LIN {X 0,Y 525.761,Z 1147.71,A -85,B 0,C 180,E1 17885.507,E2 17885.507} C_VEL
LIN {X 0,Y 527.869,Z 1135.72,A -85,B 0,C 180,E1 17883.205,E2 17883.205} C_VEL
LIN {X 0,Y 530.322,Z 1123.021,A -85,B 0,C 180,E1 17881.027,E2 17881.027} C_VEL
LIN {X 0,Y 533.766,Z 1106.397,A -85,B 0,C 180,E1 17878.491,E2 17878.491} C_VEL
LIN {X 0,Y 537.469,Z 1088.541,A -85,B 0,C 180,E1 17876.14,E2 17876.14} C_VEL
LIN {X 0,Y 540.914,Z 1072.555,A -85,B 0,C 180,E1 17874.259,E2 17874.259} C_VEL
LIN {X 0,Y 544.546,Z 1055.798,A -85,B 0,C 180,E1 17872.489,E2 17872.489} C_VEL
LIN {X 0,Y 549.152,Z 1034.672,A -85,B 0,C 180,E1 17870.505,E2 17870.505} C_VEL
LIN {X 0,Y 553.58,Z 1013.13,A -85,B 0,C 180,E1 17868.757,E2 17868.757} C_VEL
LIN {X 0,Y 557.256,Z 994.74,A -85,B 0,C 180,E1 17867.434,E2 17867.434} C_VEL
LIN {X 0,Y 560.832,Z 975.985,A -85,B 0,C 180,E1 17866.232,E2 17866.232} C_VEL
LIN {X 0,Y 564.294,Z 956.689,A -85,B 0,C 180,E1 17865.135,E2 17865.135} C_VEL
LIN {X 0,Y 568.047,Z 934.279,A -85,B 0,C 180,E1 17864.025,E2 17864.025} C_VEL
LIN {X 0,Y 572.034,Z 907.383,A -85,B 0,C 180,E1 17862.914,E2 17862.914} C_VEL
LIN {X 0,Y 574.908,Z 884.853,A -85,B 0,C 180,E1 17862.151,E2 17862.151} C_VEL
LIN {X 0,Y 577.234,Z 863.544,A -85,B 0,C 180,E1 17861.557,E2 17861.557} C_VEL
LIN {X 0,Y 579.186,Z 841.987,A -85,B 0,C 180,E1 17861.078,E2 17861.078} C_VEL
LIN {X 0,Y 580.867,Z 815.756,A -85,B 0,C 180,E1 17860.629,E2 17860.629} C_VEL
LIN {X 0,Y 589.677,Z 592.24,A -85,B 0,C 180,E1 17857.327,E2 17857.327} C_VEL
LIN {X 0,Y 595.841,Z 445.382,A -85,B 0,C 180,E1 17855.112,E2 17855.112} C_VEL
LIN {X 0,Y 585.604,Z 429.266,A -85,B 0,C 180,E1 17853.178,E2 17853.178} C_VEL
LIN {X 0,Y 575.982,Z 415.554,A -85,B 0,C 180,E1 17851.211,E2 17851.211} C_VEL
LIN {X 0,Y 566.461,Z 402.539,A -85,B 0,C 180,E1 17849.069,E2 17849.069} C_VEL
LIN {X 0,Y 561.316,Z 396.051,A -85,B 0,C 180,E1 17847.821,E2 17847.821} C_VEL
LIN {X 0,Y 556.973,Z 390.44,A -85,B 0,C 180,E1 17846.696,E2 17846.696} C_VEL
LIN {X 0,Y 552.471,Z 384.765,A -85,B 0,C 180,E1 17845.458,E2 17845.458} C_VEL
LIN {X 0,Y 548.916,Z 380.538,A -85,B 0,C 180,E1 17844.425,E2 17844.425} C_VEL
LIN {X 0,Y 544.6,Z 375.283,A -85,B 0,C 180,E1 17843.078,E2 17843.078} C_VEL
LIN {X 0,Y 541.358,Z 372.099,A -85,B 0,C 180,E1 17842.021,E2 17842.021} C_VEL
LIN {X 0,Y 539.707,Z 369.279,A -85,B 0,C 180,E1 17841.406,E2 17841.406} C_VEL
LIN {X 0,Y 536.376,Z 366.847,A -85,B 0,C 180,E1 17840.231,E2 17840.231} C_VEL
LIN {X 0,Y 534.263,Z 363.307,A -85,B 0,C 180,E1 17839.345,E2 17839.345} C_VEL
LIN {X 0,Y 533.757,Z 362.736,A -85,B 0,C 180,E1 17839.137,E2 17839.137} C_VEL
LIN {X 0,Y 530.459,Z 360.54,A -85,B 0,C 180,E1 17837.78,E2 17837.78} C_VEL
LIN {X 0,Y 528.468,Z 357.561,A -85,B 0,C 180,E1 17836.802,E2 17836.802} C_VEL
LIN {X 0,Y 527.857,Z 356.011,A -85,B 0,C 180,E1 17836.451,E2 17836.451} C_VEL
LIN {X 0,Y 524.184,Z 354.141,A -85,B 0,C 180,E1 17834.584,E2 17834.584} C_VEL
LIN {X 0,Y 522.044,Z 350.897,A -85,B 0,C 180,E1 17833.175,E2 17833.175} C_VEL
LIN {X 0,Y 521.643,Z 349.211,A -85,B 0,C 180,E1 17832.735,E2 17832.735} C_VEL
LIN {X 0,Y 521.673,Z 349.223,A -85,B 0,C 180,E1 17829.376,E2 17829.376} C_VEL
LIN {X 0,Y 521.662,Z 349.19,A -85,B 0,C 180,E1 17826.272,E2 17826.272} C_VEL
LIN {X 0,Y 521.662,Z 349.252,A -85,B 0,C 180,E1 17822.857,E2 17822.857} C_VEL
LIN {X 0,Y 521.731,Z 349.183,A -85,B 0,C 180,E1 17819.561,E2 17819.561} C_VEL
LIN {X 0,Y 521.66,Z 349.21,A -85,B 0,C 180,E1 17816.263,E2 17816.263} C_VEL
LIN {X 0,Y 521.695,Z 349.269,A -85,B 0,C 180,E1 17812.954,E2 17812.954} C_VEL
LIN {X 0,Y 522.394,Z 351.72,A -85,B 0,C 180,E1 17812.355,E2 17812.355} C_VEL
LIN {X 0,Y 524.741,Z 354.555,A -85,B 0,C 180,E1 17810.9,E2 17810.9} C_VEL
LIN {X 0,Y 528.048,Z 356.193,A -85,B 0,C 180,E1 17809.25,E2 17809.25} C_VEL
LIN {X 0,Y 529.406,Z 359.289,A -85,B 0,C 180,E1 17808.506,E2 17808.506} C_VEL
LIN {X 0,Y 532.127,Z 361.898,A -85,B 0,C 180,E1 17807.3,E2 17807.3} C_VEL
LIN {X 0,Y 534.16,Z 363.105,A -85,B 0,C 180,E1 17806.496,E2 17806.496} C_VEL
LIN {X 0,Y 536.193,Z 366.523,A -85,B 0,C 180,E1 17805.64,E2 17805.64} C_VEL
LIN {X 0,Y 539.324,Z 369.091,A -85,B 0,C 180,E1 17804.516,E2 17804.516} C_VEL
LIN {X 0,Y 540.125,Z 369.854,A -85,B 0,C 180,E1 17804.236,E2 17804.236} C_VEL
LIN {X 0,Y 542.762,Z 373.729,A -85,B 0,C 180,E1 17803.298,E2 17803.298} C_VEL
LIN {X 0,Y 545.709,Z 376.231,A -85,B 0,C 180,E1 17802.375,E2 17802.375} C_VEL
LIN {X 0,Y 548.797,Z 380.377,A -85,B 0,C 180,E1 17801.407,E2 17801.407} C_VEL
LIN {X 0,Y 551.115,Z 382.496,A -85,B 0,C 180,E1 17800.746,E2 17800.746} C_VEL
LIN {X 0,Y 554.639,Z 386.927,A -85,B 0,C 180,E1 17799.749,E2 17799.749} C_VEL
LIN {X 0,Y 556.439,Z 388.927,A -85,B 0,C 180,E1 17799.268,E2 17799.268} C_VEL
LIN {X 0,Y 560.51,Z 393.596,A -85,B 0,C 180,E1 17798.219,E2 17798.219} C_VEL
LIN {X 0,Y 564.909,Z 399.046,A -85,B 0,C 180,E1 17797.138,E2 17797.138} C_VEL
LIN {X 0,Y 574.234,Z 410.747,A -85,B 0,C 180,E1 17795.023,E2 17795.023} C_VEL
LIN {X 0,Y 581.384,Z 420.611,A -85,B 0,C 180,E1 17793.521,E2 17793.521} C_VEL
LIN {X 0,Y 590.334,Z 433.608,A -85,B 0,C 180,E1 17791.772,E2 17791.772} C_VEL
LIN {X 0,Y 595.87,Z 442.641,A -85,B 0,C 180,E1 17790.739,E2 17790.739} C_VEL
LIN {X 0,Y 586.827,Z 657.464,A -85,B 0,C 180,E1 17787.527,E2 17787.527} C_VEL
LIN {X 0,Y 580.388,Z 818.126,A -85,B 0,C 180,E1 17785.144,E2 17785.144} C_VEL
LIN {X 0,Y 578.549,Z 843.265,A -85,B 0,C 180,E1 17784.67,E2 17784.67} C_VEL
LIN {X 0,Y 575.726,Z 870.858,A -85,B 0,C 180,E1 17783.958,E2 17783.958} C_VEL
LIN {X 0,Y 573.031,Z 892.591,A -85,B 0,C 180,E1 17783.253,E2 17783.253} C_VEL
LIN {X 0,Y 570.192,Z 912.82,A -85,B 0,C 180,E1 17782.471,E2 17782.471} C_VEL
LIN {X 0,Y 566.949,Z 933.521,A -85,B 0,C 180,E1 17781.539,E2 17781.539} C_VEL
LIN {X 0,Y 563.55,Z 953.219,A -85,B 0,C 180,E1 17780.521,E2 17780.521} C_VEL
LIN {X 0,Y 561.609,Z 960.127,A -85,B 0,C 180,E1 17780.208,E2 17780.208} C_VEL
LIN {X 0,Y 553.835,Z 977.712,A -85,B 0,C 180,E1 17779.574,E2 17779.574} C_VEL
LIN {X 0,Y 551.762,Z 984.148,A -85,B 0,C 180,E1 17779.207,E2 17779.207} C_VEL
LIN {X 0,Y 547.898,Z 1002.415,A -85,B 0,C 180,E1 17777.887,E2 17777.887} C_VEL
LIN {X 0,Y 543.458,Z 1022.804,A -85,B 0,C 180,E1 17776.228,E2 17776.228} C_VEL
LIN {X 0,Y 538.244,Z 1045.707,A -85,B 0,C 180,E1 17774.074,E2 17774.074} C_VEL
LIN {X 0,Y 534.354,Z 1062.517,A -85,B 0,C 180,E1 17772.274,E2 17772.274} C_VEL
LIN {X 0,Y 530.736,Z 1078.224,A -85,B 0,C 180,E1 17770.396,E2 17770.396} C_VEL
LIN {X 0,Y 526.924,Z 1095.053,A -85,B 0,C 180,E1 17768.145,E2 17768.145} C_VEL
LIN {X 0,Y 523.166,Z 1112.322,A -85,B 0,C 180,E1 17765.493,E2 17765.493} C_VEL
LIN {X 0,Y 520.447,Z 1125.546,A -85,B 0,C 180,E1 17763.198,E2 17763.198} C_VEL
LIN {X 0,Y 518.304,Z 1136.869,A -85,B 0,C 180,E1 17761.002,E2 17761.002} C_VEL
LIN {X 0,Y 516.4,Z 1148.029,A -85,B 0,C 180,E1 17758.571,E2 17758.571} C_VEL
LIN {X 0,Y 514.548,Z 1160.441,A -85,B 0,C 180,E1 17755.432,E2 17755.432} C_VEL
LIN {X 0,Y 513.475,Z 1169.219,A -85,B 0,C 180,E1 17752.799,E2 17752.799} C_VEL
LIN {X 0,Y 512.794,Z 1176.005,A -85,B 0,C 180,E1 17750.427,E2 17750.427} C_VEL
LIN {X 0,Y 512.354,Z 1181.938,A -85,B 0,C 180,E1 17747.959,E2 17747.959} C_VEL
LIN {X 0,Y 512.062,Z 1187.545,A -85,B 0,C 180,E1 17745.052,E2 17745.052} C_VEL
LIN {X 0,Y 511.941,Z 1191.578,A -85,B 0,C 180,E1 17742.062,E2 17742.062} C_VEL
LIN {X 0,Y 511.916,Z 1193.749,A -85,B 0,C 180,E1 17739.556,E2 17739.556} C_VEL
LIN {X 0,Y 511.911,Z 1194.759,A -85,B 0,C 180,E1 17737.181,E2 17737.181} C_VEL
LIN {X 0,Y 511.902,Z 1194.8,A -85,B 0,C 180,E1 17734.93,E2 17734.93} C_VEL
LIN {X 0,Y 511.914,Z 1193.884,A -85,B 0,C 180,E1 17732.574,E2 17732.574} C_VEL
LIN {X 0,Y 511.948,Z 1191.845,A -85,B 0,C 180,E1 17730.111,E2 17730.111} C_VEL
LIN {X 0,Y 512.038,Z 1188.251,A -85,B 0,C 180,E1 17727.313,E2 17727.313} C_VEL
LIN {X 0,Y 512.321,Z 1182.436,A -85,B 0,C 180,E1 17724.175,E2 17724.175} C_VEL
LIN {X 0,Y 512.76,Z 1176.29,A -85,B 0,C 180,E1 17721.59,E2 17721.59} C_VEL
LIN {X 0,Y 513.474,Z 1169.223,A -85,B 0,C 180,E1 17719.112,E2 17719.112} C_VEL
LIN {X 0,Y 514.472,Z 1160.962,A -85,B 0,C 180,E1 17716.627,E2 17716.627} C_VEL
LIN {X 0,Y 516.231,Z 1149.055,A -85,B 0,C 180,E1 17713.573,E2 17713.573} C_VEL
LIN {X 0,Y 518.247,Z 1137.167,A -85,B 0,C 180,E1 17710.97,E2 17710.97} C_VEL
LIN {X 0,Y 520.43,Z 1125.525,A -85,B 0,C 180,E1 17708.708,E2 17708.708} C_VEL
LIN {X 0,Y 523.27,Z 1111.869,A -85,B 0,C 180,E1 17706.342,E2 17706.342} C_VEL
LIN {X 0,Y 527.274,Z 1093.391,A -85,B 0,C 180,E1 17703.536,E2 17703.536} C_VEL
LIN {X 0,Y 530.909,Z 1077.464,A -85,B 0,C 180,E1 17701.421,E2 17701.421} C_VEL
LIN {X 0,Y 534.559,Z 1061.663,A -85,B 0,C 180,E1 17699.542,E2 17699.542} C_VEL
LIN {X 0,Y 539.256,Z 1041.498,A -85,B 0,C 180,E1 17697.409,E2 17697.409} C_VEL
LIN {X 0,Y 544.119,Z 1019.613,A -85,B 0,C 180,E1 17695.413,E2 17695.413} C_VEL
LIN {X 0,Y 548.064,Z 1001.544,A -85,B 0,C 180,E1 17693.959,E2 17693.959} C_VEL
LIN {X 0,Y 551.937,Z 983.052,A -85,B 0,C 180,E1 17692.635,E2 17692.635} C_VEL
LIN {X 0,Y 555.697,Z 964.008,A -85,B 0,C 180,E1 17691.43,E2 17691.43} C_VEL
LIN {X 0,Y 560.006,Z 940.548,A -85,B 0,C 180,E1 17690.134,E2 17690.134} C_VEL
LIN {X 0,Y 563.885,Z 915.971,A -85,B 0,C 180,E1 17688.998,E2 17688.998} C_VEL
LIN {X 0,Y 566.87,Z 895.119,A -85,B 0,C 180,E1 17688.184,E2 17688.184} C_VEL
LIN {X 0,Y 569.491,Z 874.162,A -85,B 0,C 180,E1 17687.494,E2 17687.494} C_VEL
LIN {X 0,Y 571.773,Z 852.476,A -85,B 0,C 180,E1 17686.905,E2 17686.905} C_VEL
LIN {X 0,Y 574.089,Z 825.329,A -85,B 0,C 180,E1 17686.335,E2 17686.335} C_VEL
LIN {X 0,Y 576.018,Z 780.91,A -85,B 0,C 180,E1 17685.663,E2 17685.663} C_VEL
LIN {X 0,Y 584.231,Z 560.655,A -85,B 0,C 180,E1 17682.446,E2 17682.446} C_VEL
LIN {X 0,Y 588.645,Z 446.135,A -85,B 0,C 180,E1 17680.742,E2 17680.742} C_VEL
LIN {X 0,Y 571.02,Z 420.614,A -85,B 0,C 180,E1 17677.734,E2 17677.734} C_VEL
LIN {X 0,Y 561.488,Z 408.03,A -85,B 0,C 180,E1 17675.96,E2 17675.96} C_VEL
LIN {X 0,Y 552.936,Z 397.243,A -85,B 0,C 180,E1 17674.253,E2 17674.253} C_VEL
LIN {X 0,Y 548.26,Z 391.475,A -85,B 0,C 180,E1 17673.264,E2 17673.264} C_VEL
LIN {X 0,Y 544.255,Z 386.546,A -85,B 0,C 180,E1 17672.381,E2 17672.381} C_VEL
LIN {X 0,Y 539.839,Z 381.182,A -85,B 0,C 180,E1 17671.364,E2 17671.364} C_VEL
LIN {X 0,Y 536.158,Z 376.858,A -85,B 0,C 180,E1 17670.482,E2 17670.482} C_VEL
LIN {X 0,Y 534.966,Z 375.343,A -85,B 0,C 180,E1 17670.184,E2 17670.184} C_VEL
LIN {X 0,Y 531.495,Z 371.631,A -85,B 0,C 180,E1 17669.315,E2 17669.315} C_VEL
LIN {X 0,Y 529.9,Z 369.383,A -85,B 0,C 180,E1 17668.885,E2 17668.885} C_VEL
LIN {X 0,Y 526.557,Z 366.145,A -85,B 0,C 180,E1 17668.003,E2 17668.003} C_VEL
LIN {X 0,Y 524.719,Z 363.213,A -85,B 0,C 180,E1 17667.461,E2 17667.461} C_VEL
LIN {X 0,Y 521.414,Z 360.538,A -85,B 0,C 180,E1 17666.54,E2 17666.54} C_VEL
LIN {X 0,Y 519.476,Z 357.042,A -85,B 0,C 180,E1 17665.908,E2 17665.908} C_VEL
LIN {X 0,Y 515.824,Z 354.574,A -85,B 0,C 180,E1 17664.814,E2 17664.814} C_VEL
LIN {X 0,Y 514.112,Z 351.727,A -85,B 0,C 180,E1 17664.212,E2 17664.212} C_VEL
LIN {X 0,Y 513.765,Z 350.215,A -85,B 0,C 180,E1 17664.017,E2 17664.017} C_VEL
LIN {X 0,Y 513.798,Z 350.151,A -85,B 0,C 180,E1 17660.625,E2 17660.625} C_VEL
LIN {X 0,Y 513.787,Z 350.233,A -85,B 0,C 180,E1 17657.15,E2 17657.15} C_VEL
LIN {X 0,Y 513.745,Z 350.152,A -85,B 0,C 180,E1 17653.736,E2 17653.736} C_VEL
LIN {X 0,Y 513.79,Z 350.234,A -85,B 0,C 180,E1 17650.314,E2 17650.314} C_VEL
LIN {X 0,Y 513.767,Z 350.234,A -85,B 0,C 180,E1 17646.999,E2 17646.999} C_VEL
LIN {X 0,Y 513.743,Z 350.238,A -85,B 0,C 180,E1 17643.571,E2 17643.571} C_VEL
LIN {X 0,Y 513.796,Z 350.226,A -85,B 0,C 180,E1 17640.223,E2 17640.223} C_VEL
LIN {X 0,Y 513.747,Z 350.231,A -85,B 0,C 180,E1 17636.876,E2 17636.876} C_VEL
LIN {X 0,Y 513.731,Z 350.234,A -85,B 0,C 180,E1 17633.406,E2 17633.406} C_VEL
LIN {X 0,Y 513.788,Z 350.224,A -85,B 0,C 180,E1 17630.139,E2 17630.139} C_VEL
LIN {X 0,Y 513.716,Z 350.164,A -85,B 0,C 180,E1 17626.837,E2 17626.837} C_VEL
LIN {X 0,Y 513.721,Z 350.242,A -85,B 0,C 180,E1 17623.256,E2 17623.256} C_VEL
LIN {X 0,Y 513.803,Z 350.41,A -85,B 0,C 180,E1 17622.034,E2 17622.034} C_VEL
LIN {X 0,Y 514.804,Z 353.275,A -85,B 0,C 180,E1 17621.631,E2 17621.631} C_VEL
LIN {X 0,Y 517.159,Z 355.808,A -85,B 0,C 180,E1 17620.87,E2 17620.87} C_VEL
LIN {X 0,Y 519.5,Z 357.171,A -85,B 0,C 180,E1 17620.185,E2 17620.185} C_VEL
LIN {X 0,Y 521.376,Z 360.616,A -85,B 0,C 180,E1 17619.571,E2 17619.571} C_VEL
LIN {X 0,Y 524.285,Z 363.051,A -85,B 0,C 180,E1 17618.755,E2 17618.755} C_VEL
LIN {X 0,Y 525.119,Z 363.758,A -85,B 0,C 180,E1 17618.527,E2 17618.527} C_VEL
LIN {X 0,Y 527.678,Z 367.626,A -85,B 0,C 180,E1 17617.788,E2 17617.788} C_VEL
LIN {X 0,Y 530.678,Z 370.269,A -85,B 0,C 180,E1 17617.015,E2 17617.015} C_VEL
LIN {X 0,Y 533.824,Z 374.393,A -85,B 0,C 180,E1 17616.194,E2 17616.194} C_VEL
LIN {X 0,Y 535.842,Z 376.372,A -85,B 0,C 180,E1 17615.703,E2 17615.703} C_VEL
LIN {X 0,Y 539.468,Z 380.812,A -85,B 0,C 180,E1 17614.826,E2 17614.826} C_VEL
LIN {X 0,Y 548.179,Z 392.031,A -85,B 0,C 180,E1 17612.841,E2 17612.841} C_VEL
LIN {X 0,Y 557.613,Z 404.61,A -85,B 0,C 180,E1 17610.867,E2 17610.867} C_VEL
LIN {X 0,Y 568.004,Z 419.104,A -85,B 0,C 180,E1 17608.862,E2 17608.862} C_VEL
LIN {X 0,Y 578.642,Z 434.507,A -85,B 0,C 180,E1 17606.963,E2 17606.963} C_VEL
LIN {X 0,Y 588.727,Z 449.63,A -85,B 0,C 180,E1 17605.282,E2 17605.282} C_VEL
LIN {X 0,Y 580.428,Z 665.627,A -85,B 0,C 180,E1 17602.1,E2 17602.1} C_VEL
LIN {X 0,Y 574.396,Z 825.945,A -85,B 0,C 180,E1 17599.753,E2 17599.753} C_VEL
LIN {X 0,Y 572.587,Z 850.931,A -85,B 0,C 180,E1 17599.291,E2 17599.291} C_VEL
LIN {X 0,Y 569.74,Z 879.117,A -85,B 0,C 180,E1 17598.579,E2 17598.579} C_VEL
LIN {X 0,Y 567.081,Z 900.684,A -85,B 0,C 180,E1 17597.891,E2 17597.891} C_VEL
LIN {X 0,Y 564.224,Z 921.047,A -85,B 0,C 180,E1 17597.117,E2 17597.117} C_VEL
LIN {X 0,Y 560.996,Z 941.562,A -85,B 0,C 180,E1 17596.207,E2 17596.207} C_VEL
LIN {X 0,Y 556.997,Z 964.706,A -85,B 0,C 180,E1 17595.014,E2 17595.014} C_VEL
LIN {X 0,Y 552.173,Z 989.793,A -85,B 0,C 180,E1 17593.481,E2 17593.481} C_VEL
LIN {X 0,Y 548.272,Z 1008.652,A -85,B 0,C 180,E1 17592.154,E2 17592.154} C_VEL
LIN {X 0,Y 544.322,Z 1026.988,A -85,B 0,C 180,E1 17590.701,E2 17590.701} C_VEL
LIN {X 0,Y 540.247,Z 1045.394,A -85,B 0,C 180,E1 17589.064,E2 17589.064} C_VEL
LIN {X 0,Y 535.329,Z 1067.372,A -85,B 0,C 180,E1 17586.839,E2 17586.839} C_VEL
LIN {X 0,Y 531.263,Z 1085.188,A -85,B 0,C 180,E1 17584.769,E2 17584.769} C_VEL
LIN {X 0,Y 528.055,Z 1099.499,A -85,B 0,C 180,E1 17582.918,E2 17582.918} C_VEL
LIN {X 0,Y 525.032,Z 1113.285,A -85,B 0,C 180,E1 17580.944,E2 17580.944} C_VEL
LIN {X 0,Y 522.122,Z 1127.161,A -85,B 0,C 180,E1 17578.73,E2 17578.73} C_VEL
LIN {X 0,Y 519.004,Z 1143.111,A -85,B 0,C 180,E1 17575.811,E2 17575.811} C_VEL
LIN {X 0,Y 516.93,Z 1154.734,A -85,B 0,C 180,E1 17573.361,E2 17573.361} C_VEL
LIN {X 0,Y 515.375,Z 1164.513,A -85,B 0,C 180,E1 17571.034,E2 17571.034} C_VEL
LIN {X 0,Y 514.148,Z 1173.506,A -85,B 0,C 180,E1 17568.599,E2 17568.599} C_VEL
LIN {X 0,Y 513.09,Z 1183.01,A -85,B 0,C 180,E1 17565.601,E2 17565.601} C_VEL
LIN {X 0,Y 512.439,Z 1190.44,A -85,B 0,C 180,E1 17562.676,E2 17562.676} C_VEL
LIN {X 0,Y 512.138,Z 1195.692,A -85,B 0,C 180,E1 17560.121,E2 17560.121} C_VEL
LIN {X 0,Y 511.987,Z 1199.677,A -85,B 0,C 180,E1 17557.632,E2 17557.632} C_VEL
LIN {X 0,Y 511.926,Z 1202.768,A -85,B 0,C 180,E1 17554.93,E2 17554.93} C_VEL
LIN {X 0,Y 511.91,Z 1204.622,A -85,B 0,C 180,E1 17551.903,E2 17551.903} C_VEL
LIN {X 0,Y 511.897,Z 1204.871,A -85,B 0,C 180,E1 17549.329,E2 17549.329} C_VEL
LIN {X 0,Y 511.916,Z 1204.032,A -85,B 0,C 180,E1 17546.865,E2 17546.865} C_VEL
LIN {X 0,Y 511.936,Z 1202.085,A -85,B 0,C 180,E1 17544.396,E2 17544.396} C_VEL
LIN {X 0,Y 512.01,Z 1199.038,A -85,B 0,C 180,E1 17541.918,E2 17541.918} C_VEL
LIN {X 0,Y 512.197,Z 1194.454,A -85,B 0,C 180,E1 17539.199,E2 17539.199} C_VEL
LIN {X 0,Y 512.7,Z 1187.27,A -85,B 0,C 180,E1 17536.006,E2 17536.006} C_VEL
LIN {X 0,Y 513.354,Z 1180.209,A -85,B 0,C 180,E1 17533.479,E2 17533.479} C_VEL
LIN {X 0,Y 514.301,Z 1172.293,A -85,B 0,C 180,E1 17531.055,E2 17531.055} C_VEL
LIN {X 0,Y 515.578,Z 1163.145,A -85,B 0,C 180,E1 17528.618,E2 17528.618} C_VEL
LIN {X 0,Y 517.641,Z 1150.764,A -85,B 0,C 180,E1 17525.746,E2 17525.746} C_VEL
LIN {X 0,Y 520.149,Z 1136.988,A -85,B 0,C 180,E1 17523.022,E2 17523.022} C_VEL
LIN {X 0,Y 522.702,Z 1124.358,A -85,B 0,C 180,E1 17520.805,E2 17520.805} C_VEL
LIN {X 0,Y 525.619,Z 1110.662,A -85,B 0,C 180,E1 17518.665,E2 17518.665} C_VEL
LIN {X 0,Y 529.598,Z 1092.624,A -85,B 0,C 180,E1 17516.155,E2 17516.155} C_VEL
LIN {X 0,Y 533.769,Z 1073.974,A -85,B 0,C 180,E1 17513.905,E2 17513.905} C_VEL
LIN {X 0,Y 537.501,Z 1057.5,A -85,B 0,C 180,E1 17512.13,E2 17512.13} C_VEL
LIN {X 0,Y 541.483,Z 1039.846,A -85,B 0,C 180,E1 17510.428,E2 17510.428} C_VEL
LIN {X 0,Y 546.452,Z 1017.438,A -85,B 0,C 180,E1 17508.52,E2 17508.52} C_VEL
LIN {X 0,Y 551.03,Z 995.494,A -85,B 0,C 180,E1 17506.908,E2 17506.908} C_VEL
LIN {X 0,Y 554.813,Z 976.631,A -85,B 0,C 180,E1 17505.683,E2 17505.683} C_VEL
LIN {X 0,Y 558.419,Z 957.479,A -85,B 0,C 180,E1 17504.58,E2 17504.58} C_VEL
LIN {X 0,Y 562.047,Z 936.748,A -85,B 0,C 180,E1 17503.537,E2 17503.537} C_VEL
LIN {X 0,Y 566.1,Z 911.435,A -85,B 0,C 180,E1 17502.452,E2 17502.452} C_VEL
LIN {X 0,Y 569.515,Z 885.803,A -85,B 0,C 180,E1 17501.567,E2 17501.567} C_VEL
LIN {X 0,Y 571.987,Z 864.091,A -85,B 0,C 180,E1 17500.956,E2 17500.956} C_VEL
LIN {X 0,Y 574.008,Z 842.736,A -85,B 0,C 180,E1 17500.477,E2 17500.477} C_VEL
LIN {X 0,Y 575.632,Z 818.917,A -85,B 0,C 180,E1 17500.061,E2 17500.061} C_VEL
LIN {X 0,Y 584.809,Z 597.316,A -85,B 0,C 180,E1 17496.763,E2 17496.763} C_VEL
LIN {X 0,Y 591.271,Z 449.583,A -85,B 0,C 180,E1 17494.524,E2 17494.524} C_VEL
LIN {X 0,Y 581.939,Z 434.884,A -85,B 0,C 180,E1 17492.709,E2 17492.709} C_VEL
LIN {X 0,Y 571.047,Z 419.127,A -85,B 0,C 180,E1 17490.4,E2 17490.4} C_VEL
LIN {X 0,Y 562.156,Z 407.26,A -85,B 0,C 180,E1 17488.322,E2 17488.322} C_VEL
LIN {X 0,Y 558.847,Z 402.983,A -85,B 0,C 180,E1 17487.491,E2 17487.491} C_VEL
LIN {X 0,Y 554.657,Z 397.509,A -85,B 0,C 180,E1 17486.383,E2 17486.383} C_VEL
LIN {X 0,Y 550.307,Z 391.951,A -85,B 0,C 180,E1 17485.162,E2 17485.162} C_VEL
LIN {X 0,Y 546.802,Z 387.771,A -85,B 0,C 180,E1 17484.123,E2 17484.123} C_VEL
LIN {X 0,Y 542.864,Z 382.874,A -85,B 0,C 180,E1 17482.87,E2 17482.87} C_VEL
LIN {X 0,Y 539.52,Z 379.475,A -85,B 0,C 180,E1 17481.756,E2 17481.756} C_VEL
LIN {X 0,Y 537.872,Z 376.873,A -85,B 0,C 180,E1 17481.14,E2 17481.14} C_VEL
LIN {X 0,Y 534.483,Z 374.086,A -85,B 0,C 180,E1 17479.906,E2 17479.906} C_VEL
LIN {X 0,Y 532.284,Z 370.521,A -85,B 0,C 180,E1 17478.964,E2 17478.964} C_VEL
LIN {X 0,Y 528.92,Z 368.119,A -85,B 0,C 180,E1 17477.549,E2 17477.549} C_VEL
LIN {X 0,Y 526.864,Z 364.936,A -85,B 0,C 180,E1 17476.511,E2 17476.511} C_VEL
LIN {X 0,Y 526.344,Z 363.814,A -85,B 0,C 180,E1 17476.216,E2 17476.216} C_VEL
LIN {X 0,Y 522.855,Z 361.86,A -85,B 0,C 180,E1 17474.395,E2 17474.395} C_VEL
LIN {X 0,Y 520.689,Z 358.459,A -85,B 0,C 180,E1 17472.928,E2 17472.928} C_VEL
LIN {X 0,Y 520.246,Z 357.081,A -85,B 0,C 180,E1 17472.544,E2 17472.544} C_VEL
LIN {X 0,Y 515.936,Z 354.845,A -85,B 0,C 180,E1 17468.919,E2 17468.919} C_VEL
LIN {X 0,Y 513.745,Z 350.203,A -85,B 0,C 180,E1 17464.018,E2 17464.018} C_VEL
LIN {X 0,Y 513.785,Z 350.382,A -85,B 0,C 180,E1 17461.338,E2 17461.338} C_VEL
LIN {X 0,Y 516.981,Z 355.659,A -85,B 0,C 180,E1 17455.785,E2 17455.785} C_VEL
LIN {X 0,Y 520.368,Z 357.276,A -85,B 0,C 180,E1 17453.158,E2 17453.158} C_VEL
LIN {X 0,Y 521.544,Z 360.221,A -85,B 0,C 180,E1 17452.232,E2 17452.232} C_VEL
LIN {X 0,Y 524.566,Z 363.09,A -85,B 0,C 180,E1 17450.454,E2 17450.454} C_VEL
LIN {X 0,Y 526.561,Z 364.033,A -85,B 0,C 180,E1 17449.469,E2 17449.469} C_VEL
LIN {X 0,Y 528.298,Z 367.422,A -85,B 0,C 180,E1 17448.537,E2 17448.537} C_VEL
LIN {X 0,Y 531.68,Z 370.224,A -85,B 0,C 180,E1 17447.068,E2 17447.068} C_VEL
LIN {X 0,Y 532.585,Z 370.878,A -85,B 0,C 180,E1 17446.704,E2 17446.704} C_VEL
LIN {X 0,Y 535.069,Z 374.667,A -85,B 0,C 180,E1 17445.664,E2 17445.664} C_VEL
LIN {X 0,Y 538.408,Z 377.492,A -85,B 0,C 180,E1 17444.461,E2 17444.461} C_VEL
LIN {X 0,Y 541.325,Z 381.563,A -85,B 0,C 180,E1 17443.418,E2 17443.418} C_VEL
LIN {X 0,Y 543.921,Z 383.873,A -85,B 0,C 180,E1 17442.591,E2 17442.591} C_VEL
LIN {X 0,Y 547.153,Z 388.06,A -85,B 0,C 180,E1 17441.57,E2 17441.57} C_VEL
LIN {X 0,Y 549.267,Z 390.133,A -85,B 0,C 180,E1 17440.955,E2 17440.955} C_VEL
LIN {X 0,Y 553.13,Z 394.778,A -85,B 0,C 180,E1 17439.857,E2 17439.857} C_VEL
LIN {X 0,Y 559.299,Z 402.316,A -85,B 0,C 180,E1 17438.225,E2 17438.225} C_VEL
LIN {X 0,Y 564.38,Z 408.631,A -85,B 0,C 180,E1 17436.977,E2 17436.977} C_VEL
LIN {X 0,Y 571.561,Z 417.59,A -85,B 0,C 180,E1 17435.34,E2 17435.34} C_VEL
LIN {X 0,Y 578.945,Z 427.908,A -85,B 0,C 180,E1 17433.76,E2 17433.76} C_VEL
LIN {X 0,Y 587.918,Z 441.178,A -85,B 0,C 180,E1 17431.977,E2 17431.977} C_VEL
LIN {X 0,Y 591.305,Z 446.923,A -85,B 0,C 180,E1 17431.326,E2 17431.326} C_VEL
LIN {X 0,Y 581.92,Z 660.834,A -85,B 0,C 180,E1 17428.111,E2 17428.111} C_VEL
LIN {X 0,Y 575.333,Z 818.147,A -85,B 0,C 180,E1 17425.763,E2 17425.763} C_VEL
LIN {X 0,Y 573.443,Z 843.084,A -85,B 0,C 180,E1 17425.292,E2 17425.292} C_VEL
LIN {X 0,Y 570.511,Z 870.826,A -85,B 0,C 180,E1 17424.576,E2 17424.576} C_VEL
LIN {X 0,Y 567.673,Z 892.846,A -85,B 0,C 180,E1 17423.859,E2 17423.859} C_VEL
LIN {X 0,Y 564.72,Z 913.072,A -85,B 0,C 180,E1 17423.073,E2 17423.073} C_VEL
LIN {X 0,Y 561.441,Z 933.104,A -85,B 0,C 180,E1 17422.169,E2 17422.169} C_VEL
LIN {X 0,Y 557.158,Z 957.095,A -85,B 0,C 180,E1 17420.91,E2 17420.91} C_VEL
LIN {X 0,Y 552.365,Z 981.215,A -85,B 0,C 180,E1 17419.408,E2 17419.408} C_VEL
LIN {X 0,Y 551.762,Z 984.148,A -85,B 0,C 180,E1 17419.207,E2 17419.207} C_VEL
LIN {X 0,Y 549.68,Z 990.791,A -85,B 0,C 180,E1 17418.826,E2 17418.826} C_VEL
LIN {X 0,Y 541.119,Z 1008.34,A -85,B 0,C 180,E1 17417.969,E2 17417.969} C_VEL
LIN {X 0,Y 539.289,Z 1013.609,A -85,B 0,C 180,E1 17417.591,E2 17417.591} C_VEL
LIN {X 0,Y 534.899,Z 1032.31,A -85,B 0,C 180,E1 17415.942,E2 17415.942} C_VEL
LIN {X 0,Y 530.837,Z 1049.32,A -85,B 0,C 180,E1 17414.263,E2 17414.263} C_VEL
LIN {X 0,Y 526.71,Z 1066.456,A -85,B 0,C 180,E1 17412.369,E2 17412.369} C_VEL
LIN {X 0,Y 521.714,Z 1087.318,A -85,B 0,C 180,E1 17409.728,E2 17409.728} C_VEL
LIN {X 0,Y 518.113,Z 1102.59,A -85,B 0,C 180,E1 17407.516,E2 17407.516} C_VEL
LIN {X 0,Y 515.067,Z 1115.993,A -85,B 0,C 180,E1 17405.344,E2 17405.344} C_VEL
LIN {X 0,Y 512.009,Z 1130.599,A -85,B 0,C 180,E1 17402.68,E2 17402.68} C_VEL
LIN {X 0,Y 509.356,Z 1144.355,A -85,B 0,C 180,E1 17399.778,E2 17399.778} C_VEL
LIN {X 0,Y 507.627,Z 1154.545,A -85,B 0,C 180,E1 17397.318,E2 17397.318} C_VEL
LIN {X 0,Y 506.313,Z 1163.429,A -85,B 0,C 180,E1 17394.874,E2 17394.874} C_VEL
LIN {X 0,Y 505.226,Z 1172.546,A -85,B 0,C 180,E1 17391.965,E2 17391.965} C_VEL
LIN {X 0,Y 504.508,Z 1180.15,A -85,B 0,C 180,E1 17388.967,E2 17388.967} C_VEL
LIN {X 0,Y 504.173,Z 1185.477,A -85,B 0,C 180,E1 17386.356,E2 17386.356} C_VEL
LIN {X 0,Y 504.004,Z 1189.422,A -85,B 0,C 180,E1 17383.889,E2 17383.889} C_VEL
LIN {X 0,Y 503.932,Z 1192.306,A -85,B 0,C 180,E1 17381.424,E2 17381.424} C_VEL
LIN {X 0,Y 503.913,Z 1194.239,A -85,B 0,C 180,E1 17378.788,E2 17378.788} C_VEL
LIN {X 0,Y 503.896,Z 1194.955,A -85,B 0,C 180,E1 17375.693,E2 17375.693} C_VEL
LIN {X 0,Y 503.911,Z 1194.141,A -85,B 0,C 180,E1 17372.957,E2 17372.957} C_VEL
LIN {X 0,Y 503.936,Z 1192.275,A -85,B 0,C 180,E1 17370.454,E2 17370.454} C_VEL
LIN {X 0,Y 504.005,Z 1189.328,A -85,B 0,C 180,E1 17367.953,E2 17367.953} C_VEL
LIN {X 0,Y 504.174,Z 1185.291,A -85,B 0,C 180,E1 17365.45,E2 17365.45} C_VEL
LIN {X 0,Y 504.609,Z 1179.147,A -85,B 0,C 180,E1 17362.485,E2 17362.485} C_VEL
LIN {X 0,Y 505.399,Z 1170.897,A -85,B 0,C 180,E1 17359.397,E2 17359.397} C_VEL
LIN {X 0,Y 506.399,Z 1162.876,A -85,B 0,C 180,E1 17356.875,E2 17356.875} C_VEL
LIN {X 0,Y 507.695,Z 1154.046,A -85,B 0,C 180,E1 17354.464,E2 17354.464} C_VEL
LIN {X 0,Y 509.592,Z 1143.001,A -85,B 0,C 180,E1 17351.821,E2 17351.821} C_VEL
LIN {X 0,Y 512.381,Z 1128.517,A -85,B 0,C 180,E1 17348.837,E2 17348.837} C_VEL
LIN {X 0,Y 515.088,Z 1115.892,A -85,B 0,C 180,E1 17346.55,E2 17346.55} C_VEL
LIN {X 0,Y 518.121,Z 1102.538,A -85,B 0,C 180,E1 17344.387,E2 17344.387} C_VEL
LIN {X 0,Y 521.596,Z 1087.704,A -85,B 0,C 180,E1 17342.236,E2 17342.236} C_VEL
LIN {X 0,Y 526.591,Z 1066.938,A -85,B 0,C 180,E1 17339.6,E2 17339.6} C_VEL
LIN {X 0,Y 530.807,Z 1049.395,A -85,B 0,C 180,E1 17337.658,E2 17337.658} C_VEL
LIN {X 0,Y 534.923,Z 1032.152,A -85,B 0,C 180,E1 17335.956,E2 17335.956} C_VEL
LIN {X 0,Y 539.543,Z 1012.419,A -85,B 0,C 180,E1 17334.226,E2 17334.226} C_VEL
LIN {X 0,Y 544.872,Z 988.24,A -85,B 0,C 180,E1 17332.399,E2 17332.399} C_VEL
LIN {X 0,Y 548.692,Z 969.698,A -85,B 0,C 180,E1 17331.18,E2 17331.18} C_VEL
LIN {X 0,Y 552.324,Z 950.721,A -85,B 0,C 180,E1 17330.077,E2 17330.077} C_VEL
LIN {X 0,Y 555.944,Z 930.247,A -85,B 0,C 180,E1 17329.038,E2 17329.038} C_VEL
LIN {X 0,Y 559.342,Z 909.082,A -85,B 0,C 180,E1 17328.112,E2 17328.112} C_VEL
LIN {X 0,Y 563.169,Z 881.609,A -85,B 0,C 180,E1 17327.117,E2 17327.117} C_VEL
LIN {X 0,Y 565.899,Z 857.457,A -85,B 0,C 180,E1 17326.426,E2 17326.426} C_VEL
LIN {X 0,Y 567.899,Z 835.869,A -85,B 0,C 180,E1 17325.936,E2 17325.936} C_VEL
LIN {X 0,Y 569.431,Z 813.48,A -85,B 0,C 180,E1 17325.541,E2 17325.541} C_VEL
LIN {X 0,Y 577.922,Z 595.395,A -85,B 0,C 180,E1 17322.335,E2 17322.335} C_VEL
LIN {X 0,Y 583.68,Z 450.191,A -85,B 0,C 180,E1 17320.164,E2 17320.164} C_VEL
LIN {X 0,Y 566.18,Z 424.847,A -85,B 0,C 180,E1 17317.092,E2 17317.092} C_VEL
LIN {X 0,Y 554.857,Z 409.947,A -85,B 0,C 180,E1 17314.901,E2 17314.901} C_VEL
LIN {X 0,Y 545.686,Z 398.515,A -85,B 0,C 180,E1 17312.971,E2 17312.971} C_VEL
LIN {X 0,Y 541.507,Z 393.379,A -85,B 0,C 180,E1 17312.033,E2 17312.033} C_VEL
LIN {X 0,Y 537.245,Z 388.187,A -85,B 0,C 180,E1 17311.034,E2 17311.034} C_VEL
LIN {X 0,Y 533.43,Z 383.458,A -85,B 0,C 180,E1 17310.094,E2 17310.094} C_VEL
LIN {X 0,Y 529.021,Z 378.533,A -85,B 0,C 180,E1 17308.969,E2 17308.969} C_VEL
LIN {X 0,Y 527.619,Z 376.675,A -85,B 0,C 180,E1 17308.588,E2 17308.588} C_VEL
LIN {X 0,Y 524.154,Z 373.056,A -85,B 0,C 180,E1 17307.648,E2 17307.648} C_VEL
LIN {X 0,Y 522.493,Z 370.608,A -85,B 0,C 180,E1 17307.156,E2 17307.156} C_VEL
LIN {X 0,Y 519.089,Z 367.485,A -85,B 0,C 180,E1 17306.175,E2 17306.175} C_VEL
LIN {X 0,Y 517.146,Z 364.352,A -85,B 0,C 180,E1 17305.542,E2 17305.542} C_VEL
LIN {X 0,Y 513.908,Z 361.958,A -85,B 0,C 180,E1 17304.545,E2 17304.545} C_VEL
LIN {X 0,Y 511.887,Z 358.613,A -85,B 0,C 180,E1 17303.819,E2 17303.819} C_VEL
LIN {X 0,Y 511.53,Z 357.911,A -85,B 0,C 180,E1 17303.684,E2 17303.684} C_VEL
LIN {X 0,Y 508.206,Z 355.917,A -85,B 0,C 180,E1 17302.561,E2 17302.561} C_VEL
LIN {X 0,Y 506.336,Z 353.17,A -85,B 0,C 180,E1 17301.824,E2 17301.824} C_VEL
LIN {X 0,Y 505.823,Z 351.156,A -85,B 0,C 180,E1 17301.542,E2 17301.542} C_VEL
LIN {X 0,Y 505.821,Z 351.194,A -85,B 0,C 180,E1 17297.961,E2 17297.961} C_VEL
LIN {X 0,Y 505.862,Z 351.138,A -85,B 0,C 180,E1 17294.539,E2 17294.539} C_VEL
LIN {X 0,Y 505.835,Z 351.202,A -85,B 0,C 180,E1 17291.054,E2 17291.054} C_VEL
LIN {X 0,Y 505.807,Z 351.214,A -85,B 0,C 180,E1 17287.611,E2 17287.611} C_VEL
LIN {X 0,Y 505.852,Z 351.204,A -85,B 0,C 180,E1 17284.308,E2 17284.308} C_VEL
LIN {X 0,Y 505.817,Z 351.207,A -85,B 0,C 180,E1 17280.906,E2 17280.906} C_VEL
LIN {X 0,Y 505.797,Z 351.21,A -85,B 0,C 180,E1 17277.507,E2 17277.507} C_VEL
LIN {X 0,Y 505.848,Z 351.203,A -85,B 0,C 180,E1 17274.1,E2 17274.1} C_VEL
LIN {X 0,Y 505.796,Z 351.209,A -85,B 0,C 180,E1 17270.786,E2 17270.786} C_VEL
LIN {X 0,Y 505.779,Z 351.157,A -85,B 0,C 180,E1 17267.324,E2 17267.324} C_VEL
LIN {X 0,Y 505.817,Z 351.361,A -85,B 0,C 180,E1 17264.537,E2 17264.537} C_VEL
LIN {X 0,Y 506.732,Z 353.995,A -85,B 0,C 180,E1 17264.11,E2 17264.11} C_VEL
LIN {X 0,Y 508.949,Z 356.663,A -85,B 0,C 180,E1 17263.273,E2 17263.273} C_VEL
LIN {X 0,Y 511.748,Z 358.219,A -85,B 0,C 180,E1 17262.342,E2 17262.342} C_VEL
LIN {X 0,Y 513.559,Z 361.634,A -85,B 0,C 180,E1 17261.673,E2 17261.673} C_VEL
LIN {X 0,Y 516.392,Z 364.013,A -85,B 0,C 180,E1 17260.781,E2 17260.781} C_VEL
LIN {X 0,Y 517.436,Z 364.73,A -85,B 0,C 180,E1 17260.47,E2 17260.47} C_VEL
LIN {X 0,Y 519.701,Z 368.367,A -85,B 0,C 180,E1 17259.738,E2 17259.738} C_VEL
LIN {X 0,Y 523.035,Z 371.299,A -85,B 0,C 180,E1 17258.79,E2 17258.79} C_VEL
LIN {X 0,Y 525.961,Z 375.351,A -85,B 0,C 180,E1 17257.947,E2 17257.947} C_VEL
LIN {X 0,Y 528.541,Z 377.742,A -85,B 0,C 180,E1 17257.269,E2 17257.269} C_VEL
LIN {X 0,Y 532.069,Z 382.112,A -85,B 0,C 180,E1 17256.345,E2 17256.345} C_VEL
LIN {X 0,Y 533.846,Z 384.124,A -85,B 0,C 180,E1 17255.901,E2 17255.901} C_VEL
LIN {X 0,Y 541.887,Z 394.143,A -85,B 0,C 180,E1 17253.976,E2 17253.976} C_VEL
LIN {X 0,Y 553.341,Z 409.405,A -85,B 0,C 180,E1 17251.478,E2 17251.478} C_VEL
LIN {X 0,Y 564.139,Z 424.636,A -85,B 0,C 180,E1 17249.335,E2 17249.335} C_VEL
LIN {X 0,Y 575.016,Z 440.487,A -85,B 0,C 180,E1 17247.351,E2 17247.351} C_VEL
LIN {X 0,Y 583.793,Z 453.835,A -85,B 0,C 180,E1 17245.851,E2 17245.851} C_VEL
LIN {X 0,Y 575.165,Z 670.173,A -85,B 0,C 180,E1 17242.65,E2 17242.65} C_VEL
LIN {X 0,Y 569.082,Z 825.936,A -85,B 0,C 180,E1 17240.356,E2 17240.356} C_VEL
LIN {X 0,Y 567.202,Z 851.141,A -85,B 0,C 180,E1 17239.889,E2 17239.889} C_VEL
LIN {X 0,Y 564.261,Z 879.261,A -85,B 0,C 180,E1 17239.175,E2 17239.175} C_VEL
LIN {X 0,Y 561.519,Z 900.817,A -85,B 0,C 180,E1 17238.484,E2 17238.484} C_VEL
LIN {X 0,Y 558.495,Z 921.651,A -85,B 0,C 180,E1 17237.688,E2 17237.688} C_VEL
LIN {X 0,Y 555.134,Z 942.284,A -85,B 0,C 180,E1 17236.766,E2 17236.766} C_VEL
LIN {X 0,Y 550.649,Z 967.378,A -85,B 0,C 180,E1 17235.456,E2 17235.456} C_VEL
LIN {X 0,Y 546.006,Z 990.391,A -85,B 0,C 180,E1 17234.025,E2 17234.025} C_VEL
LIN {X 0,Y 541.972,Z 1009.249,A -85,B 0,C 180,E1 17232.688,E2 17232.688} C_VEL
LIN {X 0,Y 537.876,Z 1027.553,A -85,B 0,C 180,E1 17231.223,E2 17231.223} C_VEL
LIN {X 0,Y 533.498,Z 1046.511,A -85,B 0,C 180,E1 17229.516,E2 17229.516} C_VEL
LIN {X 0,Y 528.312,Z 1068.551,A -85,B 0,C 180,E1 17227.24,E2 17227.24} C_VEL
LIN {X 0,Y 524.374,Z 1085.088,A -85,B 0,C 180,E1 17225.294,E2 17225.294} C_VEL
LIN {X 0,Y 520.955,Z 1099.61,A -85,B 0,C 180,E1 17223.393,E2 17223.393} C_VEL
LIN {X 0,Y 517.661,Z 1113.962,A -85,B 0,C 180,E1 17221.305,E2 17221.305} C_VEL
LIN {X 0,Y 514.2,Z 1129.895,A -85,B 0,C 180,E1 17218.705,E2 17218.705} C_VEL
LIN {X 0,Y 511.239,Z 1144.255,A -85,B 0,C 180,E1 17215.983,E2 17215.983} C_VEL
LIN {X 0,Y 509.183,Z 1155.247,A -85,B 0,C 180,E1 17213.616,E2 17213.616} C_VEL
LIN {X 0,Y 507.546,Z 1164.97,A -85,B 0,C 180,E1 17211.253,E2 17211.253} C_VEL
LIN {X 0,Y 506.208,Z 1174.315,A -85,B 0,C 180,E1 17208.663,E2 17208.663} C_VEL
LIN {X 0,Y 505.05,Z 1184.234,A -85,B 0,C 180,E1 17205.384,E2 17205.384} C_VEL
LIN {X 0,Y 504.454,Z 1190.808,A -85,B 0,C 180,E1 17202.71,E2 17202.71} C_VEL
LIN {X 0,Y 504.146,Z 1195.895,A -85,B 0,C 180,E1 17200.167,E2 17200.167} C_VEL
LIN {X 0,Y 503.99,Z 1199.833,A -85,B 0,C 180,E1 17197.639,E2 17197.639} C_VEL
LIN {X 0,Y 503.922,Z 1202.992,A -85,B 0,C 180,E1 17194.781,E2 17194.781} C_VEL
LIN {X 0,Y 503.908,Z 1204.644,A -85,B 0,C 180,E1 17191.82,E2 17191.82} C_VEL
LIN {X 0,Y 503.901,Z 1204.848,A -85,B 0,C 180,E1 17189.205,E2 17189.205} C_VEL
LIN {X 0,Y 503.916,Z 1204.029,A -85,B 0,C 180,E1 17186.816,E2 17186.816} C_VEL
LIN {X 0,Y 503.937,Z 1202.196,A -85,B 0,C 180,E1 17184.421,E2 17184.421} C_VEL
LIN {X 0,Y 504.008,Z 1199.354,A -85,B 0,C 180,E1 17182.018,E2 17182.018} C_VEL
LIN {X 0,Y 504.166,Z 1195.484,A -85,B 0,C 180,E1 17179.603,E2 17179.603} C_VEL
LIN {X 0,Y 504.523,Z 1190.047,A -85,B 0,C 180,E1 17176.943,E2 17176.943} C_VEL
LIN {X 0,Y 505.267,Z 1181.974,A -85,B 0,C 180,E1 17173.798,E2 17173.798} C_VEL
LIN {X 0,Y 506.326,Z 1173.402,A -85,B 0,C 180,E1 17171.073,E2 17171.073} C_VEL
LIN {X 0,Y 507.614,Z 1164.519,A -85,B 0,C 180,E1 17168.63,E2 17168.63} C_VEL
LIN {X 0,Y 509.278,Z 1154.743,A -85,B 0,C 180,E1 17166.267,E2 17166.267} C_VEL
LIN {X 0,Y 511.857,Z 1141.399,A -85,B 0,C 180,E1 17163.428,E2 17163.428} C_VEL
LIN {X 0,Y 514.951,Z 1126.188,A -85,B 0,C 180,E1 17160.673,E2 17160.673} C_VEL
LIN {X 0,Y 517.837,Z 1113.179,A -85,B 0,C 180,E1 17158.579,E2 17158.579} C_VEL
LIN {X 0,Y 520.998,Z 1099.385,A -85,B 0,C 180,E1 17156.579,E2 17156.579} C_VEL
LIN {X 0,Y 524.589,Z 1084.133,A -85,B 0,C 180,E1 17154.59,E2 17154.59} C_VEL
LIN {X 0,Y 529.358,Z 1064.085,A -85,B 0,C 180,E1 17152.267,E2 17152.267} C_VEL
LIN {X 0,Y 534.02,Z 1044.123,A -85,B 0,C 180,E1 17150.266,E2 17150.266} C_VEL
LIN {X 0,Y 538.257,Z 1025.807,A -85,B 0,C 180,E1 17148.633,E2 17148.633} C_VEL
LIN {X 0,Y 542.821,Z 1005.658,A -85,B 0,C 180,E1 17147.037,E2 17147.037} C_VEL
LIN {X 0,Y 548.185,Z 980.73,A -85,B 0,C 180,E1 17145.328,E2 17145.328} C_VEL
LIN {X 0,Y 552.235,Z 960.28,A -85,B 0,C 180,E1 17144.119,E2 17144.119} C_VEL
LIN {X 0,Y 555.899,Z 940.405,A -85,B 0,C 180,E1 17143.093,E2 17143.093} C_VEL
LIN {X 0,Y 559.323,Z 920.137,A -85,B 0,C 180,E1 17142.186,E2 17142.186} C_VEL
LIN {X 0,Y 562.565,Z 898.74,A -85,B 0,C 180,E1 17141.368,E2 17141.368} C_VEL
LIN {X 0,Y 566.042,Z 872.298,A -85,B 0,C 180,E1 17140.54,E2 17140.54} C_VEL
LIN {X 0,Y 568.639,Z 846.57,A -85,B 0,C 180,E1 17139.926,E2 17139.926} C_VEL
LIN {X 0,Y 570.352,Z 824.097,A -85,B 0,C 180,E1 17139.515,E2 17139.515} C_VEL
LIN {X 0,Y 579.726,Z 608.722,A -85,B 0,C 180,E1 17136.284,E2 17136.284} C_VEL
LIN {X 0,Y 586.748,Z 453.88,A -85,B 0,C 180,E1 17133.925,E2 17133.925} C_VEL
LIN {X 0,Y 577.782,Z 439.612,A -85,B 0,C 180,E1 17132.122,E2 17132.122} C_VEL
LIN {X 0,Y 567.506,Z 424.861,A -85,B 0,C 180,E1 17129.88,E2 17129.88} C_VEL
LIN {X 0,Y 559.859,Z 414.432,A -85,B 0,C 180,E1 17128.045,E2 17128.045} C_VEL
LIN {X 0,Y 552.717,Z 404.987,A -85,B 0,C 180,E1 17126.165,E2 17126.165} C_VEL
LIN {X 0,Y 548.16,Z 399.135,A -85,B 0,C 180,E1 17124.863,E2 17124.863} C_VEL
LIN {X 0,Y 544.705,Z 394.987,A -85,B 0,C 180,E1 17123.819,E2 17123.819} C_VEL
LIN {X 0,Y 541.136,Z 390.459,A -85,B 0,C 180,E1 17122.66,E2 17122.66} C_VEL
LIN {X 0,Y 537.625,Z 386.749,A -85,B 0,C 180,E1 17121.464,E2 17121.464} C_VEL
LIN {X 0,Y 536.051,Z 384.433,A -85,B 0,C 180,E1 17120.871,E2 17120.871} C_VEL
LIN {X 0,Y 532.738,Z 381.475,A -85,B 0,C 180,E1 17119.631,E2 17119.631} C_VEL
LIN {X 0,Y 530.818,Z 378.294,A -85,B 0,C 180,E1 17118.791,E2 17118.791} C_VEL
LIN {X 0,Y 527.39,Z 375.694,A -85,B 0,C 180,E1 17117.317,E2 17117.317} C_VEL
LIN {X 0,Y 525.234,Z 372.208,A -85,B 0,C 180,E1 17116.194,E2 17116.194} C_VEL
LIN {X 0,Y 524.733,Z 371.552,A -85,B 0,C 180,E1 17115.926,E2 17115.926} C_VEL
LIN {X 0,Y 521.354,Z 369.388,A -85,B 0,C 180,E1 17114.097,E2 17114.097} C_VEL
LIN {X 0,Y 519.344,Z 366.02,A -85,B 0,C 180,E1 17112.679,E2 17112.679} C_VEL
LIN {X 0,Y 518.962,Z 364.954,A -85,B 0,C 180,E1 17112.349,E2 17112.349} C_VEL
LIN {X 0,Y 514.689,Z 362.543,A -85,B 0,C 180,E1 17108.603,E2 17108.603} C_VEL
LIN {X 0,Y 512.735,Z 358.139,A -85,B 0,C 180,E1 17104.026,E2 17104.026} C_VEL
LIN {X 0,Y 512.788,Z 358.254,A -85,B 0,C 180,E1 17101.453,E2 17101.453} C_VEL
LIN {X 0,Y 516.004,Z 363.617,A -85,B 0,C 180,E1 17095.777,E2 17095.777} C_VEL
LIN {X 0,Y 519.101,Z 365.2,A -85,B 0,C 180,E1 17093.336,E2 17093.336} C_VEL
LIN {X 0,Y 520.55,Z 368.368,A -85,B 0,C 180,E1 17092.217,E2 17092.217} C_VEL
LIN {X 0,Y 523.805,Z 371.178,A -85,B 0,C 180,E1 17090.329,E2 17090.329} C_VEL
LIN {X 0,Y 525.139,Z 371.89,A -85,B 0,C 180,E1 17089.662,E2 17089.662} C_VEL
LIN {X 0,Y 527.195,Z 375.508,A -85,B 0,C 180,E1 17088.568,E2 17088.568} C_VEL
LIN {X 0,Y 531.081,Z 378.71,A -85,B 0,C 180,E1 17086.887,E2 17086.887} C_VEL
LIN {X 0,Y 533.952,Z 382.765,A -85,B 0,C 180,E1 17085.689,E2 17085.689} C_VEL
LIN {X 0,Y 536.703,Z 385.1,A -85,B 0,C 180,E1 17084.687,E2 17084.687} C_VEL
LIN {X 0,Y 539.74,Z 389.24,A -85,B 0,C 180,E1 17083.59,E2 17083.59} C_VEL
LIN {X 0,Y 542.145,Z 391.488,A -85,B 0,C 180,E1 17082.809,E2 17082.809} C_VEL
LIN {X 0,Y 545.681,Z 395.895,A -85,B 0,C 180,E1 17081.684,E2 17081.684} C_VEL
LIN {X 0,Y 547.429,Z 397.749,A -85,B 0,C 180,E1 17081.165,E2 17081.165} C_VEL
LIN {X 0,Y 551.443,Z 402.461,A -85,B 0,C 180,E1 17080.014,E2 17080.014} C_VEL
LIN {X 0,Y 556.097,Z 408.124,A -85,B 0,C 180,E1 17078.758,E2 17078.758} C_VEL
LIN {X 0,Y 565.863,Z 420.56,A -85,B 0,C 180,E1 17076.352,E2 17076.352} C_VEL
LIN {X 0,Y 573.988,Z 431.415,A -85,B 0,C 180,E1 17074.542,E2 17074.542} C_VEL
LIN {X 0,Y 584.279,Z 446.828,A -85,B 0,C 180,E1 17072.425,E2 17072.425} C_VEL
LIN {X 0,Y 586.815,Z 451.112,A -85,B 0,C 180,E1 17071.924,E2 17071.924} C_VEL
LIN {X 0,Y 577.078,Z 664.425,A -85,B 0,C 180,E1 17068.703,E2 17068.703} C_VEL
LIN {X 0,Y 570.36,Z 818.193,A -85,B 0,C 180,E1 17066.394,E2 17066.394} C_VEL
LIN {X 0,Y 568.385,Z 843.364,A -85,B 0,C 180,E1 17065.916,E2 17065.916} C_VEL
LIN {X 0,Y 565.34,Z 871.1,A -85,B 0,C 180,E1 17065.198,E2 17065.198} C_VEL
LIN {X 0,Y 562.491,Z 892.492,A -85,B 0,C 180,E1 17064.501,E2 17064.501} C_VEL
LIN {X 0,Y 559.427,Z 912.739,A -85,B 0,C 180,E1 17063.714,E2 17063.714} C_VEL
LIN {X 0,Y 556.019,Z 932.774,A -85,B 0,C 180,E1 17062.809,E2 17062.809} C_VEL
LIN {X 0,Y 551.946,Z 954.65,A -85,B 0,C 180,E1 17061.664,E2 17061.664} C_VEL
LIN {X 0,Y 546.617,Z 980.683,A -85,B 0,C 180,E1 17060.054,E2 17060.054} C_VEL
LIN {X 0,Y 542.247,Z 1000.5,A -85,B 0,C 180,E1 17058.632,E2 17058.632} C_VEL
LIN {X 0,Y 539.289,Z 1013.609,A -85,B 0,C 180,E1 17057.591,E2 17057.591} C_VEL
LIN {X 0,Y 537.043,Z 1019.803,A -85,B 0,C 180,E1 17057.142,E2 17057.142} C_VEL
LIN {X 0,Y 528.584,Z 1035.605,A -85,B 0,C 180,E1 17056.159,E2 17056.159} C_VEL
LIN {X 0,Y 526.389,Z 1041.414,A -85,B 0,C 180,E1 17055.662,E2 17055.662} C_VEL
LIN {X 0,Y 521.322,Z 1061.358,A -85,B 0,C 180,E1 17053.515,E2 17053.515} C_VEL
LIN {X 0,Y 517.437,Z 1076.704,A -85,B 0,C 180,E1 17051.661,E2 17051.661} C_VEL
LIN {X 0,Y 513.739,Z 1091.494,A -85,B 0,C 180,E1 17049.67,E2 17049.67} C_VEL
LIN {X 0,Y 509.892,Z 1107.246,A -85,B 0,C 180,E1 17047.295,E2 17047.295} C_VEL
LIN {X 0,Y 506.025,Z 1123.861,A -85,B 0,C 180,E1 17044.41,E2 17044.41} C_VEL
LIN {X 0,Y 503.363,Z 1136.088,A -85,B 0,C 180,E1 17041.983,E2 17041.983} C_VEL
LIN {X 0,Y 501.2,Z 1147.099,A -85,B 0,C 180,E1 17039.521,E2 17039.521} C_VEL
LIN {X 0,Y 499.212,Z 1158.872,A -85,B 0,C 180,E1 17036.528,E2 17036.528} C_VEL
LIN {X 0,Y 497.782,Z 1168.592,A -85,B 0,C 180,E1 17033.56,E2 17033.56} C_VEL
LIN {X 0,Y 496.966,Z 1175.78,A -85,B 0,C 180,E1 17030.985,E2 17030.985} C_VEL
LIN {X 0,Y 496.425,Z 1181.751,A -85,B 0,C 180,E1 17028.434,E2 17028.434} C_VEL
LIN {X 0,Y 496.121,Z 1186.984,A -85,B 0,C 180,E1 17025.667,E2 17025.667} C_VEL
LIN {X 0,Y 495.953,Z 1191.38,A -85,B 0,C 180,E1 17022.457,E2 17022.457} C_VEL
LIN {X 0,Y 495.914,Z 1193.698,A -85,B 0,C 180,E1 17019.75,E2 17019.75} C_VEL
LIN {X 0,Y 495.914,Z 1194.744,A -85,B 0,C 180,E1 17017.297,E2 17017.297} C_VEL
LIN {X 0,Y 495.903,Z 1194.815,A -85,B 0,C 180,E1 17014.973,E2 17014.973} C_VEL
LIN {X 0,Y 495.914,Z 1193.923,A -85,B 0,C 180,E1 17012.542,E2 17012.542} C_VEL
LIN {X 0,Y 495.949,Z 1192.028,A -85,B 0,C 180,E1 17010.115,E2 17010.115} C_VEL
LIN {X 0,Y 496.027,Z 1188.984,A -85,B 0,C 180,E1 17007.573,E2 17007.573} C_VEL
LIN {X 0,Y 496.24,Z 1184.442,A -85,B 0,C 180,E1 17004.797,E2 17004.797} C_VEL
LIN {X 0,Y 496.798,Z 1177.382,A -85,B 0,C 180,E1 17001.551,E2 17001.551} C_VEL
LIN {X 0,Y 497.598,Z 1170.156,A -85,B 0,C 180,E1 16998.877,E2 16998.877} C_VEL
LIN {X 0,Y 498.631,Z 1162.426,A -85,B 0,C 180,E1 16996.431,E2 16996.431} C_VEL
LIN {X 0,Y 500.053,Z 1153.537,A -85,B 0,C 180,E1 16993.982,E2 16993.982} C_VEL
LIN {X 0,Y 502.419,Z 1140.914,A -85,B 0,C 180,E1 16990.95,E2 16990.95} C_VEL
LIN {X 0,Y 505.229,Z 1127.295,A -85,B 0,C 180,E1 16988.155,E2 16988.155} C_VEL
LIN {X 0,Y 507.993,Z 1115.215,A -85,B 0,C 180,E1 16985.956,E2 16985.956} C_VEL
LIN {X 0,Y 511.181,Z 1101.785,A -85,B 0,C 180,E1 16983.764,E2 16983.764} C_VEL
LIN {X 0,Y 515.515,Z 1084.424,A -85,B 0,C 180,E1 16981.247,E2 16981.247} C_VEL
LIN {X 0,Y 520.281,Z 1065.429,A -85,B 0,C 180,E1 16978.871,E2 16978.871} C_VEL
LIN {X 0,Y 524.331,Z 1049.318,A -85,B 0,C 180,E1 16977.079,E2 16977.079} C_VEL
LIN {X 0,Y 528.479,Z 1032.631,A -85,B 0,C 180,E1 16975.417,E2 16975.417} C_VEL
LIN {X 0,Y 532.801,Z 1014.736,A -85,B 0,C 180,E1 16973.828,E2 16973.828} C_VEL
LIN {X 0,Y 538.309,Z 990.953,A -85,B 0,C 180,E1 16971.987,E2 16971.987} C_VEL
LIN {X 0,Y 542.737,Z 970.142,A -85,B 0,C 180,E1 16970.604,E2 16970.604} C_VEL
LIN {X 0,Y 546.495,Z 951.161,A -85,B 0,C 180,E1 16969.495,E2 16969.495} C_VEL
LIN {X 0,Y 550.042,Z 931.756,A -85,B 0,C 180,E1 16968.5,E2 16968.5} C_VEL
LIN {X 0,Y 553.339,Z 912.014,A -85,B 0,C 180,E1 16967.623,E2 16967.623} C_VEL
LIN {X 0,Y 556.55,Z 890.449,A -85,B 0,C 180,E1 16966.804,E2 16966.804} C_VEL
LIN {X 0,Y 559.964,Z 863.517,A -85,B 0,C 180,E1 16965.969,E2 16965.969} C_VEL
LIN {X 0,Y 562.414,Z 838.278,A -85,B 0,C 180,E1 16965.37,E2 16965.37} C_VEL
LIN {X 0,Y 564.05,Z 815.956,A -85,B 0,C 180,E1 16964.966,E2 16964.966} C_VEL
LIN {X 0,Y 572.476,Z 608.164,A -85,B 0,C 180,E1 16961.892,E2 16961.892} C_VEL
LIN {X 0,Y 578.875,Z 454.526,A -85,B 0,C 180,E1 16959.596,E2 16959.596} C_VEL
LIN {X 0,Y 562.709,Z 430.981,A -85,B 0,C 180,E1 16956.691,E2 16956.691} C_VEL
LIN {X 0,Y 551.864,Z 416.584,A -85,B 0,C 180,E1 16954.549,E2 16954.549} C_VEL
LIN {X 0,Y 542.802,Z 405.177,A -85,B 0,C 180,E1 16952.603,E2 16952.603} C_VEL
LIN {X 0,Y 538.78,Z 400.199,A -85,B 0,C 180,E1 16951.682,E2 16951.682} C_VEL
LIN {X 0,Y 534.774,Z 395.268,A -85,B 0,C 180,E1 16950.724,E2 16950.724} C_VEL
LIN {X 0,Y 530.112,Z 389.617,A -85,B 0,C 180,E1 16949.554,E2 16949.554} C_VEL
LIN {X 0,Y 526.384,Z 385.153,A -85,B 0,C 180,E1 16948.569,E2 16948.569} C_VEL
LIN {X 0,Y 521.598,Z 379.702,A -85,B 0,C 180,E1 16947.238,E2 16947.238} C_VEL
LIN {X 0,Y 520.288,Z 377.948,A -85,B 0,C 180,E1 16946.848,E2 16946.848} C_VEL
LIN {X 0,Y 516.787,Z 374.418,A -85,B 0,C 180,E1 16945.807,E2 16945.807} C_VEL
LIN {X 0,Y 515.181,Z 371.902,A -85,B 0,C 180,E1 16945.277,E2 16945.277} C_VEL
LIN {X 0,Y 511.847,Z 369.156,A -85,B 0,C 180,E1 16944.22,E2 16944.22} C_VEL
LIN {X 0,Y 509.631,Z 365.568,A -85,B 0,C 180,E1 16943.41,E2 16943.41} C_VEL
LIN {X 0,Y 506.235,Z 363.183,A -85,B 0,C 180,E1 16942.225,E2 16942.225} C_VEL
LIN {X 0,Y 504.288,Z 360.073,A -85,B 0,C 180,E1 16941.428,E2 16941.428} C_VEL
LIN {X 0,Y 503.732,Z 358.861,A -85,B 0,C 180,E1 16941.178,E2 16941.178} C_VEL
LIN {X 0,Y 500.265,Z 356.909,A -85,B 0,C 180,E1 16939.803,E2 16939.803} C_VEL
LIN {X 0,Y 498.442,Z 354.151,A -85,B 0,C 180,E1 16938.934,E2 16938.934} C_VEL
LIN {X 0,Y 497.921,Z 352.151,A -85,B 0,C 180,E1 16938.589,E2 16938.589} C_VEL
LIN {X 0,Y 497.886,Z 352.144,A -85,B 0,C 180,E1 16935.253,E2 16935.253} C_VEL
LIN {X 0,Y 497.87,Z 352.163,A -85,B 0,C 180,E1 16931.703,E2 16931.703} C_VEL
LIN {X 0,Y 497.913,Z 352.189,A -85,B 0,C 180,E1 16928.313,E2 16928.313} C_VEL
LIN {X 0,Y 497.876,Z 352.192,A -85,B 0,C 180,E1 16925.054,E2 16925.054} C_VEL
LIN {X 0,Y 497.864,Z 352.194,A -85,B 0,C 180,E1 16921.611,E2 16921.611} C_VEL
LIN {X 0,Y 497.917,Z 352.188,A -85,B 0,C 180,E1 16918.274,E2 16918.274} C_VEL
LIN {X 0,Y 497.867,Z 352.195,A -85,B 0,C 180,E1 16914.815,E2 16914.815} C_VEL
LIN {X 0,Y 497.849,Z 352.197,A -85,B 0,C 180,E1 16911.336,E2 16911.336} C_VEL
LIN {X 0,Y 497.892,Z 352.151,A -85,B 0,C 180,E1 16907.945,E2 16907.945} C_VEL
LIN {X 0,Y 497.873,Z 352.321,A -85,B 0,C 180,E1 16907.502,E2 16907.502} C_VEL
LIN {X 0,Y 498.705,Z 354.898,A -85,B 0,C 180,E1 16907.023,E2 16907.023} C_VEL
LIN {X 0,Y 501.051,Z 357.553,A -85,B 0,C 180,E1 16905.968,E2 16905.968} C_VEL
LIN {X 0,Y 503.927,Z 359.108,A -85,B 0,C 180,E1 16904.846,E2 16904.846} C_VEL
LIN {X 0,Y 505.782,Z 362.7,A -85,B 0,C 180,E1 16904.05,E2 16904.05} C_VEL
LIN {X 0,Y 508.463,Z 365.049,A -85,B 0,C 180,E1 16903.08,E2 16903.08} C_VEL
LIN {X 0,Y 509.887,Z 365.958,A -85,B 0,C 180,E1 16902.599,E2 16902.599} C_VEL
LIN {X 0,Y 512.098,Z 369.541,A -85,B 0,C 180,E1 16901.796,E2 16901.796} C_VEL
LIN {X 0,Y 515.512,Z 372.389,A -85,B 0,C 180,E1 16900.718,E2 16900.718} C_VEL
LIN {X 0,Y 518.205,Z 376.275,A -85,B 0,C 180,E1 16899.853,E2 16899.853} C_VEL
LIN {X 0,Y 520.971,Z 378.764,A -85,B 0,C 180,E1 16899.055,E2 16899.055} C_VEL
LIN {X 0,Y 524.248,Z 383.065,A -85,B 0,C 180,E1 16898.107,E2 16898.107} C_VEL
LIN {X 0,Y 526.419,Z 385.177,A -85,B 0,C 180,E1 16897.526,E2 16897.526} C_VEL
LIN {X 0,Y 530.119,Z 389.643,A -85,B 0,C 180,E1 16896.548,E2 16896.548} C_VEL
LIN {X 0,Y 538.813,Z 400.385,A -85,B 0,C 180,E1 16894.41,E2 16894.41} C_VEL
LIN {X 0,Y 550.662,Z 416.438,A -85,B 0,C 180,E1 16891.77,E2 16891.77} C_VEL
LIN {X 0,Y 561.243,Z 431.519,A -85,B 0,C 180,E1 16889.634,E2 16889.634} C_VEL
LIN {X 0,Y 571.9,Z 447.243,A -85,B 0,C 180,E1 16887.656,E2 16887.656} C_VEL
LIN {X 0,Y 578.915,Z 457.974,A -85,B 0,C 180,E1 16886.431,E2 16886.431} C_VEL
LIN {X 0,Y 569.933,Z 675.046,A -85,B 0,C 180,E1 16883.203,E2 16883.203} C_VEL
LIN {X 0,Y 563.819,Z 825.913,A -85,B 0,C 180,E1 16880.969,E2 16880.969} C_VEL
LIN {X 0,Y 561.847,Z 851.582,A -85,B 0,C 180,E1 16880.491,E2 16880.491} C_VEL
LIN {X 0,Y 558.831,Z 879.401,A -85,B 0,C 180,E1 16879.78,E2 16879.78} C_VEL
LIN {X 0,Y 556.03,Z 900.779,A -85,B 0,C 180,E1 16879.094,E2 16879.094} C_VEL
LIN {X 0,Y 552.969,Z 921.2,A -85,B 0,C 180,E1 16878.313,E2 16878.313} C_VEL
LIN {X 0,Y 549.545,Z 941.611,A -85,B 0,C 180,E1 16877.402,E2 16877.402} C_VEL
LIN {X 0,Y 545.054,Z 965.995,A -85,B 0,C 180,E1 16876.133,E2 16876.133} C_VEL
LIN {X 0,Y 540.058,Z 990.091,A -85,B 0,C 180,E1 16874.638,E2 16874.638} C_VEL
LIN {X 0,Y 535.951,Z 1008.714,A -85,B 0,C 180,E1 16873.314,E2 16873.314} C_VEL
LIN {X 0,Y 531.79,Z 1026.723,A -85,B 0,C 180,E1 16871.873,E2 16871.873} C_VEL
LIN {X 0,Y 527.516,Z 1044.568,A -85,B 0,C 180,E1 16870.267,E2 16870.267} C_VEL
LIN {X 0,Y 522.495,Z 1065.123,A -85,B 0,C 180,E1 16868.179,E2 16868.179} C_VEL
LIN {X 0,Y 517.638,Z 1084.523,A -85,B 0,C 180,E1 16865.891,E2 16865.891} C_VEL
LIN {X 0,Y 513.988,Z 1099.302,A -85,B 0,C 180,E1 16863.939,E2 16863.939} C_VEL
LIN {X 0,Y 510.677,Z 1113.09,A -85,B 0,C 180,E1 16861.914,E2 16861.914} C_VEL
LIN {X 0,Y 507.441,Z 1126.979,A -85,B 0,C 180,E1 16859.642,E2 16859.642} C_VEL
LIN {X 0,Y 503.845,Z 1143.614,A -85,B 0,C 180,E1 16856.52,E2 16856.52} C_VEL
LIN {X 0,Y 501.607,Z 1154.889,A -85,B 0,C 180,E1 16854.081,E2 16854.081} C_VEL
LIN {X 0,Y 499.879,Z 1164.51,A -85,B 0,C 180,E1 16851.719,E2 16851.719} C_VEL
LIN {X 0,Y 498.546,Z 1173.098,A -85,B 0,C 180,E1 16849.325,E2 16849.325} C_VEL
LIN {X 0,Y 497.418,Z 1181.619,A -85,B 0,C 180,E1 16846.585,E2 16846.585} C_VEL
LIN {X 0,Y 496.6,Z 1189.788,A -85,B 0,C 180,E1 16843.389,E2 16843.389} C_VEL
LIN {X 0,Y 496.198,Z 1195.273,A -85,B 0,C 180,E1 16840.684,E2 16840.684} C_VEL
LIN {X 0,Y 496.018,Z 1199.234,A -85,B 0,C 180,E1 16838.198,E2 16838.198} C_VEL
LIN {X 0,Y 495.939,Z 1202.08,A -85,B 0,C 180,E1 16835.786,E2 16835.786} C_VEL
LIN {X 0,Y 495.916,Z 1203.958,A -85,B 0,C 180,E1 16833.352,E2 16833.352} C_VEL
LIN {X 0,Y 495.906,Z 1204.826,A -85,B 0,C 180,E1 16830.925,E2 16830.925} C_VEL
LIN {X 0,Y 495.91,Z 1204.712,A -85,B 0,C 180,E1 16828.498,E2 16828.498} C_VEL
LIN {X 0,Y 495.919,Z 1203.413,A -85,B 0,C 180,E1 16825.722,E2 16825.722} C_VEL
LIN {X 0,Y 495.988,Z 1200.31,A -85,B 0,C 180,E1 16822.588,E2 16822.588} C_VEL
LIN {X 0,Y 496.144,Z 1196.307,A -85,B 0,C 180,E1 16819.903,E2 16819.903} C_VEL
LIN {X 0,Y 496.456,Z 1191.316,A -85,B 0,C 180,E1 16817.319,E2 16817.319} C_VEL
LIN {X 0,Y 497.003,Z 1185.445,A -85,B 0,C 180,E1 16814.839,E2 16814.839} C_VEL
LIN {X 0,Y 497.897,Z 1177.735,A -85,B 0,C 180,E1 16812.107,E2 16812.107} C_VEL
LIN {X 0,Y 499.522,Z 1166.783,A -85,B 0,C 180,E1 16808.875,E2 16808.875} C_VEL
LIN {X 0,Y 501.326,Z 1156.414,A -85,B 0,C 180,E1 16806.273,E2 16806.273} C_VEL
LIN {X 0,Y 503.235,Z 1146.507,A -85,B 0,C 180,E1 16804.08,E2 16804.08} C_VEL
LIN {X 0,Y 505.674,Z 1134.945,A -85,B 0,C 180,E1 16801.799,E2 16801.799} C_VEL
LIN {X 0,Y 508.725,Z 1121.328,A -85,B 0,C 180,E1 16799.4,E2 16799.4} C_VEL
LIN {X 0,Y 513.172,Z 1102.679,A -85,B 0,C 180,E1 16796.537,E2 16796.537} C_VEL
LIN {X 0,Y 516.944,Z 1087.283,A -85,B 0,C 180,E1 16794.464,E2 16794.464} C_VEL
LIN {X 0,Y 520.674,Z 1072.221,A -85,B 0,C 180,E1 16792.64,E2 16792.64} C_VEL
LIN {X 0,Y 524.662,Z 1056.161,A -85,B 0,C 180,E1 16790.891,E2 16790.891} C_VEL
LIN {X 0,Y 529.651,Z 1036.031,A -85,B 0,C 180,E1 16788.933,E2 16788.933} C_VEL
LIN {X 0,Y 535.098,Z 1013.066,A -85,B 0,C 180,E1 16786.998,E2 16786.998} C_VEL
LIN {X 0,Y 539.634,Z 993.28,A -85,B 0,C 180,E1 16785.543,E2 16785.543} C_VEL
LIN {X 0,Y 543.717,Z 974.591,A -85,B 0,C 180,E1 16784.328,E2 16784.328} C_VEL
LIN {X 0,Y 547.608,Z 955.575,A -85,B 0,C 180,E1 16783.237,E2 16783.237} C_VEL
LIN {X 0,Y 552.077,Z 931.807,A -85,B 0,C 180,E1 16782.051,E2 16782.051} C_VEL
LIN {X 0,Y 556.315,Z 905.862,A -85,B 0,C 180,E1 16780.986,E2 16780.986} C_VEL
LIN {X 0,Y 559.412,Z 884.187,A -85,B 0,C 180,E1 16780.253,E2 16780.253} C_VEL
LIN {X 0,Y 561.983,Z 863.003,A -85,B 0,C 180,E1 16779.661,E2 16779.661} C_VEL
LIN {X 0,Y 564.138,Z 841.487,A -85,B 0,C 180,E1 16779.183,E2 16779.183} C_VEL
LIN {X 0,Y 566.057,Z 814.157,A -85,B 0,C 180,E1 16778.711,E2 16778.711} C_VEL
LIN {X 0,Y 576.137,Z 589.083,A -85,B 0,C 180,E1 16775.328,E2 16775.328} C_VEL
LIN {X 0,Y 582.368,Z 458.204,A -85,B 0,C 180,E1 16773.327,E2 16773.327} C_VEL
LIN {X 0,Y 573.256,Z 443.815,A -85,B 0,C 180,E1 16771.435,E2 16771.435} C_VEL
LIN {X 0,Y 562.075,Z 427.617,A -85,B 0,C 180,E1 16768.88,E2 16768.88} C_VEL
LIN {X 0,Y 554.335,Z 417.298,A -85,B 0,C 180,E1 16766.92,E2 16766.92} C_VEL
LIN {X 0,Y 549.994,Z 411.524,A -85,B 0,C 180,E1 16765.725,E2 16765.725} C_VEL
LIN {X 0,Y 546.197,Z 406.511,A -85,B 0,C 180,E1 16764.612,E2 16764.612} C_VEL
LIN {X 0,Y 542.467,Z 402.014,A -85,B 0,C 180,E1 16763.462,E2 16763.462} C_VEL
LIN {X 0,Y 539.259,Z 397.919,A -85,B 0,C 180,E1 16762.398,E2 16762.398} C_VEL
LIN {X 0,Y 535.743,Z 394.022,A -85,B 0,C 180,E1 16761.17,E2 16761.17} C_VEL
LIN {X 0,Y 534.536,Z 392.152,A -85,B 0,C 180,E1 16760.704,E2 16760.704} C_VEL
LIN {X 0,Y 531.145,Z 389.047,A -85,B 0,C 180,E1 16759.412,E2 16759.412} C_VEL
LIN {X 0,Y 529.098,Z 385.923,A -85,B 0,C 180,E1 16758.511,E2 16758.511} C_VEL
LIN {X 0,Y 525.65,Z 383.007,A -85,B 0,C 180,E1 16756.977,E2 16756.977} C_VEL
LIN {X 0,Y 523.57,Z 379.441,A -85,B 0,C 180,E1 16755.849,E2 16755.849} C_VEL
LIN {X 0,Y 520.213,Z 377.289,A -85,B 0,C 180,E1 16754.015,E2 16754.015} C_VEL
LIN {X 0,Y 518.073,Z 373.752,A -85,B 0,C 180,E1 16752.484,E2 16752.484} C_VEL
LIN {X 0,Y 517.686,Z 372.817,A -85,B 0,C 180,E1 16752.153,E2 16752.153} C_VEL
LIN {X 0,Y 513.543,Z 370.326,A -85,B 0,C 180,E1 16748.397,E2 16748.397} C_VEL
LIN {X 0,Y 511.74,Z 366.077,A -85,B 0,C 180,E1 16743.921,E2 16743.921} C_VEL
LIN {X 0,Y 511.802,Z 366.268,A -85,B 0,C 180,E1 16741.455,E2 16741.455} C_VEL
LIN {X 0,Y 515.026,Z 371.575,A -85,B 0,C 180,E1 16735.769,E2 16735.769} C_VEL
LIN {X 0,Y 517.848,Z 373.052,A -85,B 0,C 180,E1 16733.514,E2 16733.514} C_VEL
LIN {X 0,Y 519.398,Z 376.269,A -85,B 0,C 180,E1 16732.311,E2 16732.311} C_VEL
LIN {X 0,Y 522.628,Z 379.052,A -85,B 0,C 180,E1 16730.419,E2 16730.419} C_VEL
LIN {X 0,Y 523.776,Z 379.795,A -85,B 0,C 180,E1 16729.829,E2 16729.829} C_VEL
LIN {X 0,Y 525.986,Z 383.436,A -85,B 0,C 180,E1 16728.653,E2 16728.653} C_VEL
LIN {X 0,Y 529.588,Z 386.497,A -85,B 0,C 180,E1 16727.071,E2 16727.071} C_VEL
LIN {X 0,Y 532.703,Z 390.702,A -85,B 0,C 180,E1 16725.766,E2 16725.766} C_VEL
LIN {X 0,Y 535.073,Z 392.804,A -85,B 0,C 180,E1 16724.889,E2 16724.889} C_VEL
LIN {X 0,Y 538.311,Z 397.063,A -85,B 0,C 180,E1 16723.711,E2 16723.711} C_VEL
LIN {X 0,Y 540.378,Z 399.081,A -85,B 0,C 180,E1 16723.029,E2 16723.029} C_VEL
LIN {X 0,Y 544.046,Z 403.573,A -85,B 0,C 180,E1 16721.849,E2 16721.849} C_VEL
LIN {X 0,Y 545.762,Z 405.579,A -85,B 0,C 180,E1 16721.327,E2 16721.327} C_VEL
LIN {X 0,Y 550.594,Z 411.52,A -85,B 0,C 180,E1 16719.926,E2 16719.926} C_VEL
LIN {X 0,Y 555.162,Z 417.182,A -85,B 0,C 180,E1 16718.693,E2 16718.693} C_VEL
LIN {X 0,Y 560.235,Z 423.622,A -85,B 0,C 180,E1 16717.408,E2 16717.408} C_VEL
LIN {X 0,Y 566.867,Z 432.171,A -85,B 0,C 180,E1 16715.844,E2 16715.844} C_VEL
LIN {X 0,Y 574.749,Z 443.361,A -85,B 0,C 180,E1 16714.109,E2 16714.109} C_VEL
LIN {X 0,Y 582.393,Z 455.38,A -85,B 0,C 180,E1 16712.53,E2 16712.53} C_VEL
LIN {X 0,Y 572.297,Z 668.231,A -85,B 0,C 180,E1 16709.302,E2 16709.302} C_VEL
LIN {X 0,Y 565.462,Z 818.382,A -85,B 0,C 180,E1 16707.034,E2 16707.034} C_VEL
LIN {X 0,Y 563.39,Z 843.904,A -85,B 0,C 180,E1 16706.548,E2 16706.548} C_VEL
LIN {X 0,Y 560.258,Z 871.35,A -85,B 0,C 180,E1 16705.833,E2 16705.833} C_VEL
LIN {X 0,Y 557.273,Z 892.974,A -85,B 0,C 180,E1 16705.125,E2 16705.125} C_VEL
LIN {X 0,Y 553.992,Z 913.809,A -85,B 0,C 180,E1 16704.309,E2 16704.309} C_VEL
LIN {X 0,Y 550.257,Z 934.877,A -85,B 0,C 180,E1 16703.345,E2 16703.345} C_VEL
LIN {X 0,Y 545.242,Z 960.481,A -85,B 0,C 180,E1 16701.963,E2 16701.963} C_VEL
LIN {X 0,Y 540.478,Z 982.332,A -85,B 0,C 180,E1 16700.566,E2 16700.566} C_VEL
LIN {X 0,Y 536.179,Z 1001,A -85,B 0,C 180,E1 16699.21,E2 16699.21} C_VEL
LIN {X 0,Y 531.703,Z 1019.652,A -85,B 0,C 180,E1 16697.683,E2 16697.683} C_VEL
LIN {X 0,Y 526.389,Z 1041.414,A -85,B 0,C 180,E1 16695.662,E2 16695.662} C_VEL
LIN {X 0,Y 524.164,Z 1047.184,A -85,B 0,C 180,E1 16695.145,E2 16695.145} C_VEL
LIN {X 0,Y 515.031,Z 1062.616,A -85,B 0,C 180,E1 16693.891,E2 16693.891} C_VEL
LIN {X 0,Y 513.197,Z 1067.244,A -85,B 0,C 180,E1 16693.403,E2 16693.403} C_VEL
LIN {X 0,Y 507.785,Z 1087.709,A -85,B 0,C 180,E1 16690.749,E2 16690.749} C_VEL
LIN {X 0,Y 503.924,Z 1102.621,A -85,B 0,C 180,E1 16688.537,E2 16688.537} C_VEL
LIN {X 0,Y 500.673,Z 1115.635,A -85,B 0,C 180,E1 16686.379,E2 16686.379} C_VEL
LIN {X 0,Y 497.423,Z 1129.304,A -85,B 0,C 180,E1 16683.834,E2 16683.834} C_VEL
LIN {X 0,Y 494.21,Z 1144.05,A -85,B 0,C 180,E1 16680.653,E2 16680.653} C_VEL
LIN {X 0,Y 492.22,Z 1154.21,A -85,B 0,C 180,E1 16678.117,E2 16678.117} C_VEL
LIN {X 0,Y 490.72,Z 1163.125,A -85,B 0,C 180,E1 16675.592,E2 16675.592} C_VEL
LIN {X 0,Y 489.579,Z 1171.329,A -85,B 0,C 180,E1 16672.912,E2 16672.912} C_VEL
LIN {X 0,Y 488.661,Z 1179.702,A -85,B 0,C 180,E1 16669.607,E2 16669.607} C_VEL
LIN {X 0,Y 488.225,Z 1185.326,A -85,B 0,C 180,E1 16666.784,E2 16666.784} C_VEL
LIN {X 0,Y 488.022,Z 1189.306,A -85,B 0,C 180,E1 16664.232,E2 16664.232} C_VEL
LIN {X 0,Y 487.937,Z 1192.088,A -85,B 0,C 180,E1 16661.824,E2 16661.824} C_VEL
LIN {X 0,Y 487.915,Z 1193.982,A -85,B 0,C 180,E1 16659.316,E2 16659.316} C_VEL
LIN {X 0,Y 487.894,Z 1194.839,A -85,B 0,C 180,E1 16656.826,E2 16656.826} C_VEL
LIN {X 0,Y 487.912,Z 1194.675,A -85,B 0,C 180,E1 16654.23,E2 16654.23} C_VEL
LIN {X 0,Y 487.923,Z 1193.127,A -85,B 0,C 180,E1 16651.174,E2 16651.174} C_VEL
LIN {X 0,Y 487.992,Z 1190.061,A -85,B 0,C 180,E1 16648.238,E2 16648.238} C_VEL
LIN {X 0,Y 488.163,Z 1186.239,A -85,B 0,C 180,E1 16645.653,E2 16645.653} C_VEL
LIN {X 0,Y 488.511,Z 1181.34,A -85,B 0,C 180,E1 16643.077,E2 16643.077} C_VEL
LIN {X 0,Y 489.073,Z 1175.554,A -85,B 0,C 180,E1 16640.586,E2 16640.586} C_VEL
LIN {X 0,Y 490.012,Z 1168.038,A -85,B 0,C 180,E1 16637.867,E2 16637.867} C_VEL
LIN {X 0,Y 491.729,Z 1157.022,A -85,B 0,C 180,E1 16634.546,E2 16634.546} C_VEL
LIN {X 0,Y 493.6,Z 1146.918,A -85,B 0,C 180,E1 16631.945,E2 16631.945} C_VEL
LIN {X 0,Y 495.782,Z 1136.52,A -85,B 0,C 180,E1 16629.58,E2 16629.58} C_VEL
LIN {X 0,Y 498.44,Z 1124.869,A -85,B 0,C 180,E1 16627.222,E2 16627.222} C_VEL
LIN {X 0,Y 502.299,Z 1109.142,A -85,B 0,C 180,E1 16624.408,E2 16624.408} C_VEL
LIN {X 0,Y 506.523,Z 1092.505,A -85,B 0,C 180,E1 16621.849,E2 16621.849} C_VEL
LIN {X 0,Y 510.49,Z 1077.339,A -85,B 0,C 180,E1 16619.776,E2 16619.776} C_VEL
LIN {X 0,Y 514.684,Z 1061.489,A -85,B 0,C 180,E1 16617.839,E2 16617.839} C_VEL
LIN {X 0,Y 519.87,Z 1041.77,A -85,B 0,C 180,E1 16615.699,E2 16615.699} C_VEL
LIN {X 0,Y 525.257,Z 1020.273,A -85,B 0,C 180,E1 16613.699,E2 16613.699} C_VEL
LIN {X 0,Y 529.63,Z 1002.227,A -85,B 0,C 180,E1 16612.221,E2 16612.221} C_VEL
LIN {X 0,Y 533.924,Z 983.614,A -85,B 0,C 180,E1 16610.868,E2 16610.868} C_VEL
LIN {X 0,Y 538.459,Z 962.714,A -85,B 0,C 180,E1 16609.534,E2 16609.534} C_VEL
LIN {X 0,Y 543.601,Z 936.538,A -85,B 0,C 180,E1 16608.111,E2 16608.111} C_VEL
LIN {X 0,Y 547.374,Z 914.902,A -85,B 0,C 180,E1 16607.122,E2 16607.122} C_VEL
LIN {X 0,Y 550.565,Z 894.383,A -85,B 0,C 180,E1 16606.321,E2 16606.321} C_VEL
LIN {X 0,Y 553.416,Z 873.397,A -85,B 0,C 180,E1 16605.632,E2 16605.632} C_VEL
LIN {X 0,Y 556.086,Z 850.072,A -85,B 0,C 180,E1 16605.006,E2 16605.006} C_VEL
LIN {X 0,Y 558.589,Z 820.601,A -85,B 0,C 180,E1 16604.416,E2 16604.416} C_VEL
LIN {X 0,Y 561.343,Z 758.558,A -85,B 0,C 180,E1 16603.481,E2 16603.481} C_VEL
LIN {X 0,Y 570.288,Z 544.963,A -85,B 0,C 180,E1 16600.304,E2 16600.304} C_VEL
LIN {X 0,Y 573.988,Z 458.795,A -85,B 0,C 180,E1 16599,E2 16599} C_VEL
LIN {X 0,Y 559.62,Z 437.58,A -85,B 0,C 180,E1 16596.353,E2 16596.353} C_VEL
LIN {X 0,Y 548.892,Z 423.216,A -85,B 0,C 180,E1 16594.193,E2 16594.193} C_VEL
LIN {X 0,Y 539.729,Z 411.561,A -85,B 0,C 180,E1 16592.183,E2 16592.183} C_VEL
LIN {X 0,Y 535.351,Z 406.137,A -85,B 0,C 180,E1 16591.156,E2 16591.156} C_VEL
LIN {X 0,Y 532.218,Z 402.237,A -85,B 0,C 180,E1 16590.388,E2 16590.388} C_VEL
LIN {X 0,Y 527.613,Z 396.632,A -85,B 0,C 180,E1 16589.209,E2 16589.209} C_VEL
LIN {X 0,Y 522.918,Z 391.015,A -85,B 0,C 180,E1 16587.935,E2 16587.935} C_VEL
LIN {X 0,Y 519.237,Z 386.606,A -85,B 0,C 180,E1 16586.876,E2 16586.876} C_VEL
LIN {X 0,Y 517.922,Z 385.107,A -85,B 0,C 180,E1 16586.485,E2 16586.485} C_VEL
LIN {X 0,Y 514.425,Z 381.219,A -85,B 0,C 180,E1 16585.409,E2 16585.409} C_VEL
LIN {X 0,Y 513.059,Z 379.315,A -85,B 0,C 180,E1 16584.957,E2 16584.957} C_VEL
LIN {X 0,Y 509.573,Z 376.044,A -85,B 0,C 180,E1 16583.811,E2 16583.811} C_VEL
LIN {X 0,Y 507.664,Z 373.123,A -85,B 0,C 180,E1 16583.104,E2 16583.104} C_VEL
LIN {X 0,Y 504.145,Z 370.249,A -85,B 0,C 180,E1 16581.832,E2 16581.832} C_VEL
LIN {X 0,Y 501.919,Z 366.542,A -85,B 0,C 180,E1 16580.884,E2 16580.884} C_VEL
LIN {X 0,Y 498.544,Z 364.342,A -85,B 0,C 180,E1 16579.502,E2 16579.502} C_VEL
LIN {X 0,Y 496.671,Z 361.318,A -85,B 0,C 180,E1 16578.578,E2 16578.578} C_VEL
LIN {X 0,Y 496.234,Z 360.009,A -85,B 0,C 180,E1 16578.321,E2 16578.321} C_VEL
LIN {X 0,Y 492.961,Z 358.469,A -85,B 0,C 180,E1 16576.74,E2 16576.74} C_VEL
LIN {X 0,Y 490.729,Z 355.742,A -85,B 0,C 180,E1 16575.421,E2 16575.421} C_VEL
LIN {X 0,Y 489.997,Z 353.226,A -85,B 0,C 180,E1 16574.839,E2 16574.839} C_VEL
LIN {X 0,Y 489.934,Z 353.159,A -85,B 0,C 180,E1 16571.418,E2 16571.418} C_VEL
LIN {X 0,Y 489.937,Z 353.186,A -85,B 0,C 180,E1 16567.859,E2 16567.859} C_VEL
LIN {X 0,Y 489.98,Z 353.178,A -85,B 0,C 180,E1 16564.448,E2 16564.448} C_VEL
LIN {X 0,Y 489.937,Z 353.184,A -85,B 0,C 180,E1 16560.936,E2 16560.936} C_VEL
LIN {X 0,Y 489.918,Z 353.187,A -85,B 0,C 180,E1 16557.427,E2 16557.427} C_VEL
LIN {X 0,Y 489.96,Z 353.182,A -85,B 0,C 180,E1 16554.026,E2 16554.026} C_VEL
LIN {X 0,Y 489.935,Z 353.376,A -85,B 0,C 180,E1 16551.289,E2 16551.289} C_VEL
LIN {X 0,Y 490.73,Z 355.818,A -85,B 0,C 180,E1 16550.678,E2 16550.678} C_VEL
LIN {X 0,Y 493.168,Z 358.698,A -85,B 0,C 180,E1 16549.25,E2 16549.25} C_VEL
LIN {X 0,Y 496.205,Z 360.2,A -85,B 0,C 180,E1 16547.785,E2 16547.785} C_VEL
LIN {X 0,Y 497.693,Z 363.339,A -85,B 0,C 180,E1 16546.996,E2 16546.996} C_VEL
LIN {X 0,Y 500.765,Z 366.068,A -85,B 0,C 180,E1 16545.665,E2 16545.665} C_VEL
LIN {X 0,Y 502.235,Z 366.914,A -85,B 0,C 180,E1 16545.089,E2 16545.089} C_VEL
LIN {X 0,Y 504.509,Z 370.751,A -85,B 0,C 180,E1 16544.127,E2 16544.127} C_VEL
LIN {X 0,Y 507.517,Z 373.088,A -85,B 0,C 180,E1 16543.047,E2 16543.047} C_VEL
LIN {X 0,Y 508.191,Z 373.841,A -85,B 0,C 180,E1 16542.805,E2 16542.805} C_VEL
LIN {X 0,Y 510.802,Z 377.577,A -85,B 0,C 180,E1 16541.866,E2 16541.866} C_VEL
LIN {X 0,Y 513.607,Z 379.968,A -85,B 0,C 180,E1 16540.968,E2 16540.968} C_VEL
LIN {X 0,Y 516.714,Z 384.154,A -85,B 0,C 180,E1 16539.97,E2 16539.97} C_VEL
LIN {X 0,Y 519.005,Z 386.332,A -85,B 0,C 180,E1 16539.297,E2 16539.297} C_VEL
LIN {X 0,Y 522.541,Z 390.77,A -85,B 0,C 180,E1 16538.268,E2 16538.268} C_VEL
LIN {X 0,Y 524.399,Z 392.723,A -85,B 0,C 180,E1 16537.76,E2 16537.76} C_VEL
LIN {X 0,Y 529.605,Z 399.076,A -85,B 0,C 180,E1 16536.376,E2 16536.376} C_VEL
LIN {X 0,Y 536.577,Z 407.836,A -85,B 0,C 180,E1 16534.651,E2 16534.651} C_VEL
LIN {X 0,Y 547.887,Z 423.305,A -85,B 0,C 180,E1 16532.088,E2 16532.088} C_VEL
LIN {X 0,Y 558.827,Z 439.062,A -85,B 0,C 180,E1 16529.845,E2 16529.845} C_VEL
LIN {X 0,Y 569.282,Z 454.752,A -85,B 0,C 180,E1 16527.876,E2 16527.876} C_VEL
LIN {X 0,Y 574.08,Z 462.224,A -85,B 0,C 180,E1 16527.019,E2 16527.019} C_VEL
LIN {X 0,Y 564.814,Z 678.243,A -85,B 0,C 180,E1 16523.792,E2 16523.792} C_VEL
LIN {X 0,Y 558.611,Z 825.87,A -85,B 0,C 180,E1 16521.593,E2 16521.593} C_VEL
LIN {X 0,Y 556.564,Z 851.765,A -85,B 0,C 180,E1 16521.109,E2 16521.109} C_VEL
LIN {X 0,Y 553.48,Z 879.333,A -85,B 0,C 180,E1 16520.403,E2 16520.403} C_VEL
LIN {X 0,Y 550.567,Z 900.897,A -85,B 0,C 180,E1 16519.708,E2 16519.708} C_VEL
LIN {X 0,Y 547.411,Z 921.28,A -85,B 0,C 180,E1 16518.927,E2 16518.927} C_VEL
LIN {X 0,Y 543.756,Z 942.391,A -85,B 0,C 180,E1 16517.978,E2 16517.978} C_VEL
LIN {X 0,Y 538.923,Z 967.635,A -85,B 0,C 180,E1 16516.648,E2 16516.648} C_VEL
LIN {X 0,Y 533.986,Z 990.555,A -85,B 0,C 180,E1 16515.208,E2 16515.208} C_VEL
LIN {X 0,Y 529.669,Z 1009.467,A -85,B 0,C 180,E1 16513.852,E2 16513.852} C_VEL
LIN {X 0,Y 525.27,Z 1027.83,A -85,B 0,C 180,E1 16512.366,E2 16512.366} C_VEL
LIN {X 0,Y 520.397,Z 1047.465,A -85,B 0,C 180,E1 16510.571,E2 16510.571} C_VEL
LIN {X 0,Y 514.822,Z 1069.104,A -85,B 0,C 180,E1 16508.284,E2 16508.284} C_VEL
LIN {X 0,Y 510.598,Z 1085.353,A -85,B 0,C 180,E1 16506.326,E2 16506.326} C_VEL
LIN {X 0,Y 506.799,Z 1100.053,A -85,B 0,C 180,E1 16504.351,E2 16504.351} C_VEL
LIN {X 0,Y 503.13,Z 1114.697,A -85,B 0,C 180,E1 16502.155,E2 16502.155} C_VEL
LIN {X 0,Y 499.019,Z 1131.654,A -85,B 0,C 180,E1 16499.269,E2 16499.269} C_VEL
LIN {X 0,Y 496.089,Z 1144.673,A -85,B 0,C 180,E1 16496.709,E2 16496.709} C_VEL
LIN {X 0,Y 493.866,Z 1155.371,A -85,B 0,C 180,E1 16494.344,E2 16494.344} C_VEL
LIN {X 0,Y 492.078,Z 1164.962,A -85,B 0,C 180,E1 16491.955,E2 16491.955} C_VEL
LIN {X 0,Y 490.614,Z 1173.907,A -85,B 0,C 180,E1 16489.402,E2 16489.402} C_VEL
LIN {X 0,Y 489.286,Z 1183.622,A -85,B 0,C 180,E1 16486.137,E2 16486.137} C_VEL
LIN {X 0,Y 488.578,Z 1190.548,A -85,B 0,C 180,E1 16483.251,E2 16483.251} C_VEL
LIN {X 0,Y 488.207,Z 1195.476,A -85,B 0,C 180,E1 16480.742,E2 16480.742} C_VEL
LIN {X 0,Y 488.021,Z 1199.348,A -85,B 0,C 180,E1 16478.246,E2 16478.246} C_VEL
LIN {X 0,Y 487.939,Z 1202.191,A -85,B 0,C 180,E1 16475.763,E2 16475.763} C_VEL
LIN {X 0,Y 487.916,Z 1204.024,A -85,B 0,C 180,E1 16473.29,E2 16473.29} C_VEL
LIN {X 0,Y 487.898,Z 1204.871,A -85,B 0,C 180,E1 16470.705,E2 16470.705} C_VEL
LIN {X 0,Y 487.909,Z 1204.548,A -85,B 0,C 180,E1 16467.651,E2 16467.651} C_VEL
LIN {X 0,Y 487.934,Z 1202.531,A -85,B 0,C 180,E1 16464.592,E2 16464.592} C_VEL
LIN {X 0,Y 488.012,Z 1199.668,A -85,B 0,C 180,E1 16461.992,E2 16461.992} C_VEL
LIN {X 0,Y 488.189,Z 1195.824,A -85,B 0,C 180,E1 16459.459,E2 16459.459} C_VEL
LIN {X 0,Y 488.533,Z 1191.013,A -85,B 0,C 180,E1 16456.968,E2 16456.968} C_VEL
LIN {X 0,Y 489.12,Z 1185.138,A -85,B 0,C 180,E1 16454.467,E2 16454.467} C_VEL
LIN {X 0,Y 490.219,Z 1176.674,A -85,B 0,C 180,E1 16451.447,E2 16451.447} C_VEL
LIN {X 0,Y 491.835,Z 1166.351,A -85,B 0,C 180,E1 16448.41,E2 16448.41} C_VEL
LIN {X 0,Y 493.707,Z 1156.209,A -85,B 0,C 180,E1 16445.852,E2 16445.852} C_VEL
LIN {X 0,Y 495.83,Z 1145.829,A -85,B 0,C 180,E1 16443.535,E2 16443.535} C_VEL
LIN {X 0,Y 498.572,Z 1133.563,A -85,B 0,C 180,E1 16441.098,E2 16441.098} C_VEL
LIN {X 0,Y 502.407,Z 1117.621,A -85,B 0,C 180,E1 16438.305,E2 16438.305} C_VEL
LIN {X 0,Y 506.582,Z 1100.87,A -85,B 0,C 180,E1 16435.77,E2 16435.77} C_VEL
LIN {X 0,Y 510.469,Z 1085.775,A -85,B 0,C 180,E1 16433.734,E2 16433.734} C_VEL
LIN {X 0,Y 514.813,Z 1069.071,A -85,B 0,C 180,E1 16431.716,E2 16431.716} C_VEL
LIN {X 0,Y 520.666,Z 1046.619,A -85,B 0,C 180,E1 16429.338,E2 16429.338} C_VEL
LIN {X 0,Y 525.511,Z 1027.577,A -85,B 0,C 180,E1 16427.583,E2 16427.583} C_VEL
LIN {X 0,Y 529.924,Z 1009.738,A -85,B 0,C 180,E1 16426.119,E2 16426.119} C_VEL
LIN {X 0,Y 534.601,Z 990.069,A -85,B 0,C 180,E1 16424.689,E2 16424.689} C_VEL
LIN {X 0,Y 540.042,Z 965.849,A -85,B 0,C 180,E1 16423.158,E2 16423.158} C_VEL
LIN {X 0,Y 544.824,Z 941.972,A -85,B 0,C 180,E1 16421.89,E2 16421.89} C_VEL
LIN {X 0,Y 548.641,Z 921.067,A -85,B 0,C 180,E1 16420.94,E2 16420.94} C_VEL
LIN {X 0,Y 551.995,Z 900.612,A -85,B 0,C 180,E1 16420.147,E2 16420.147} C_VEL
LIN {X 0,Y 555.153,Z 878.542,A -85,B 0,C 180,E1 16419.429,E2 16419.429} C_VEL
LIN {X 0,Y 558.488,Z 850.022,A -85,B 0,C 180,E1 16418.702,E2 16418.702} C_VEL
LIN {X 0,Y 560.554,Z 825.358,A -85,B 0,C 180,E1 16418.239,E2 16418.239} C_VEL
LIN {X 0,Y 570.338,Z 618.16,A -85,B 0,C 180,E1 16415.096,E2 16415.096} C_VEL
LIN {X 0,Y 578.05,Z 462.601,A -85,B 0,C 180,E1 16412.721,E2 16412.721} C_VEL
LIN {X 0,Y 569.639,Z 449.337,A -85,B 0,C 180,E1 16410.922,E2 16410.922} C_VEL
LIN {X 0,Y 559.259,Z 434.124,A -85,B 0,C 180,E1 16408.484,E2 16408.484} C_VEL
LIN {X 0,Y 552.01,Z 424.34,A -85,B 0,C 180,E1 16406.607,E2 16406.607} C_VEL
LIN {X 0,Y 547.393,Z 418.135,A -85,B 0,C 180,E1 16405.305,E2 16405.305} C_VEL
LIN {X 0,Y 543.833,Z 413.39,A -85,B 0,C 180,E1 16404.234,E2 16404.234} C_VEL
LIN {X 0,Y 537.55,Z 405.494,A -85,B 0,C 180,E1 16402.185,E2 16402.185} C_VEL
LIN {X 0,Y 533.876,Z 401.295,A -85,B 0,C 180,E1 16400.874,E2 16400.874} C_VEL
LIN {X 0,Y 532.739,Z 399.679,A -85,B 0,C 180,E1 16400.432,E2 16400.432} C_VEL
LIN {X 0,Y 529.291,Z 396.246,A -85,B 0,C 180,E1 16399.076,E2 16399.076} C_VEL
LIN {X 0,Y 527.648,Z 393.667,A -85,B 0,C 180,E1 16398.335,E2 16398.335} C_VEL
LIN {X 0,Y 524.128,Z 390.552,A -85,B 0,C 180,E1 16396.734,E2 16396.734} C_VEL
LIN {X 0,Y 521.978,Z 387.16,A -85,B 0,C 180,E1 16395.556,E2 16395.556} C_VEL
LIN {X 0,Y 518.732,Z 384.807,A -85,B 0,C 180,E1 16393.715,E2 16393.715} C_VEL
LIN {X 0,Y 516.684,Z 381.137,A -85,B 0,C 180,E1 16392.177,E2 16392.177} C_VEL
LIN {X 0,Y 516.263,Z 380.622,A -85,B 0,C 180,E1 16391.847,E2 16391.847} C_VEL
LIN {X 0,Y 512.249,Z 377.877,A -85,B 0,C 180,E1 16387.966,E2 16387.966} C_VEL
LIN {X 0,Y 510.764,Z 374.018,A -85,B 0,C 180,E1 16383.929,E2 16383.929} C_VEL
LIN {X 0,Y 510.807,Z 374.14,A -85,B 0,C 180,E1 16381.57,E2 16381.57} C_VEL
LIN {X 0,Y 513.933,Z 379.46,A -85,B 0,C 180,E1 16375.872,E2 16375.872} C_VEL
LIN {X 0,Y 516.633,Z 380.962,A -85,B 0,C 180,E1 16373.666,E2 16373.666} C_VEL
LIN {X 0,Y 518.328,Z 384.268,A -85,B 0,C 180,E1 16372.351,E2 16372.351} C_VEL
LIN {X 0,Y 521.66,Z 387.027,A -85,B 0,C 180,E1 16370.401,E2 16370.401} C_VEL
LIN {X 0,Y 522.423,Z 387.657,A -85,B 0,C 180,E1 16369.997,E2 16369.997} C_VEL
LIN {X 0,Y 524.89,Z 391.474,A -85,B 0,C 180,E1 16368.685,E2 16368.685} C_VEL
LIN {X 0,Y 528.047,Z 394.155,A -85,B 0,C 180,E1 16367.283,E2 16367.283} C_VEL
LIN {X 0,Y 531.321,Z 398.502,A -85,B 0,C 180,E1 16365.895,E2 16365.895} C_VEL
LIN {X 0,Y 533.453,Z 400.488,A -85,B 0,C 180,E1 16365.092,E2 16365.092} C_VEL
LIN {X 0,Y 536.885,Z 404.88,A -85,B 0,C 180,E1 16363.834,E2 16363.834} C_VEL
LIN {X 0,Y 538.693,Z 406.776,A -85,B 0,C 180,E1 16363.224,E2 16363.224} C_VEL
LIN {X 0,Y 542.581,Z 411.398,A -85,B 0,C 180,E1 16361.965,E2 16361.965} C_VEL
LIN {X 0,Y 548.722,Z 419.106,A -85,B 0,C 180,E1 16360.133,E2 16360.133} C_VEL
LIN {X 0,Y 553.154,Z 424.667,A -85,B 0,C 180,E1 16358.917,E2 16358.917} C_VEL
LIN {X 0,Y 560.597,Z 434.108,A -85,B 0,C 180,E1 16357.035,E2 16357.035} C_VEL
LIN {X 0,Y 568.801,Z 445.457,A -85,B 0,C 180,E1 16355.129,E2 16355.129} C_VEL
LIN {X 0,Y 577.988,Z 459.522,A -85,B 0,C 180,E1 16353.159,E2 16353.159} C_VEL
LIN {X 0,Y 568.543,Z 651.882,A -85,B 0,C 180,E1 16350.217,E2 16350.217} C_VEL
LIN {X 0,Y 560.666,Z 818.302,A -85,B 0,C 180,E1 16347.691,E2 16347.691} C_VEL
LIN {X 0,Y 558.558,Z 843.52,A -85,B 0,C 180,E1 16347.211,E2 16347.211} C_VEL
LIN {X 0,Y 555.298,Z 871.314,A -85,B 0,C 180,E1 16346.49,E2 16346.49} C_VEL
LIN {X 0,Y 552.248,Z 892.74,A -85,B 0,C 180,E1 16345.788,E2 16345.788} C_VEL
LIN {X 0,Y 548.892,Z 913.345,A -85,B 0,C 180,E1 16344.983,E2 16344.983} C_VEL
LIN {X 0,Y 545.203,Z 933.492,A -85,B 0,C 180,E1 16344.064,E2 16344.064} C_VEL
LIN {X 0,Y 540.421,Z 957.326,A -85,B 0,C 180,E1 16342.796,E2 16342.796} C_VEL
LIN {X 0,Y 534.835,Z 982.137,A -85,B 0,C 180,E1 16341.221,E2 16341.221} C_VEL
LIN {X 0,Y 530.179,Z 1001.561,A -85,B 0,C 180,E1 16339.799,E2 16339.799} C_VEL
LIN {X 0,Y 525.455,Z 1020.415,A -85,B 0,C 180,E1 16338.238,E2 16338.238} C_VEL
LIN {X 0,Y 519.804,Z 1042.388,A -85,B 0,C 180,E1 16336.164,E2 16336.164} C_VEL
LIN {X 0,Y 514.617,Z 1061.848,A -85,B 0,C 180,E1 16334.036,E2 16334.036} C_VEL
LIN {X 0,Y 513.197,Z 1067.244,A -85,B 0,C 180,E1 16333.403,E2 16333.403} C_VEL
LIN {X 0,Y 510.959,Z 1072.609,A -85,B 0,C 180,E1 16332.825,E2 16332.825} C_VEL
LIN {X 0,Y 502.213,Z 1086.195,A -85,B 0,C 180,E1 16331.458,E2 16331.458} C_VEL
LIN {X 0,Y 500.026,Z 1091.07,A -85,B 0,C 180,E1 16330.823,E2 16330.823} C_VEL
LIN {X 0,Y 496.042,Z 1105.909,A -85,B 0,C 180,E1 16328.546,E2 16328.546} C_VEL
LIN {X 0,Y 491.463,Z 1123.543,A -85,B 0,C 180,E1 16325.438,E2 16325.438} C_VEL
LIN {X 0,Y 488.499,Z 1135.816,A -85,B 0,C 180,E1 16322.942,E2 16322.942} C_VEL
LIN {X 0,Y 486.111,Z 1146.565,A -85,B 0,C 180,E1 16320.475,E2 16320.475} C_VEL
LIN {X 0,Y 484.079,Z 1156.725,A -85,B 0,C 180,E1 16317.827,E2 16317.827} C_VEL
LIN {X 0,Y 482.167,Z 1167.965,A -85,B 0,C 180,E1 16314.372,E2 16314.372} C_VEL
LIN {X 0,Y 481.203,Z 1175.243,A -85,B 0,C 180,E1 16311.706,E2 16311.706} C_VEL
LIN {X 0,Y 480.572,Z 1181.109,A -85,B 0,C 180,E1 16309.159,E2 16309.159} C_VEL
LIN {X 0,Y 480.221,Z 1185.779,A -85,B 0,C 180,E1 16306.698,E2 16306.698} C_VEL
LIN {X 0,Y 480.024,Z 1189.492,A -85,B 0,C 180,E1 16304.228,E2 16304.228} C_VEL
LIN {X 0,Y 479.936,Z 1192.334,A -85,B 0,C 180,E1 16301.658,E2 16301.658} C_VEL
LIN {X 0,Y 479.914,Z 1194.197,A -85,B 0,C 180,E1 16298.989,E2 16298.989} C_VEL
LIN {X 0,Y 479.903,Z 1194.988,A -85,B 0,C 180,E1 16295.859,E2 16295.859} C_VEL
LIN {X 0,Y 479.911,Z 1194.166,A -85,B 0,C 180,E1 16292.866,E2 16292.866} C_VEL
LIN {X 0,Y 479.947,Z 1192.323,A -85,B 0,C 180,E1 16290.238,E2 16290.238} C_VEL
LIN {X 0,Y 480.022,Z 1189.558,A -85,B 0,C 180,E1 16287.731,E2 16287.731} C_VEL
LIN {X 0,Y 480.205,Z 1185.796,A -85,B 0,C 180,E1 16285.222,E2 16285.222} C_VEL
LIN {X 0,Y 480.588,Z 1181.021,A -85,B 0,C 180,E1 16282.708,E2 16282.708} C_VEL
LIN {X 0,Y 481.24,Z 1174.781,A -85,B 0,C 180,E1 16280.015,E2 16280.015} C_VEL
LIN {X 0,Y 482.573,Z 1165.483,A -85,B 0,C 180,E1 16276.703,E2 16276.703} C_VEL
LIN {X 0,Y 484.253,Z 1155.73,A -85,B 0,C 180,E1 16273.814,E2 16273.814} C_VEL
LIN {X 0,Y 486.217,Z 1145.946,A -85,B 0,C 180,E1 16271.288,E2 16271.288} C_VEL
LIN {X 0,Y 488.714,Z 1134.877,A -85,B 0,C 180,E1 16268.769,E2 16268.769} C_VEL
LIN {X 0,Y 492.402,Z 1119.904,A -85,B 0,C 180,E1 16265.783,E2 16265.783} C_VEL
LIN {X 0,Y 496.323,Z 1104.704,A -85,B 0,C 180,E1 16263.175,E2 16263.175} C_VEL
LIN {X 0,Y 500.055,Z 1090.854,A -85,B 0,C 180,E1 16261.06,E2 16261.06} C_VEL
LIN {X 0,Y 504.269,Z 1075.517,A -85,B 0,C 180,E1 16258.966,E2 16258.966} C_VEL
LIN {X 0,Y 509.636,Z 1056.153,A -85,B 0,C 180,E1 16256.629,E2 16256.629} C_VEL
LIN {X 0,Y 515.078,Z 1035.75,A -85,B 0,C 180,E1 16254.519,E2 16254.519} C_VEL
LIN {X 0,Y 519.503,Z 1018.693,A -85,B 0,C 180,E1 16252.956,E2 16252.956} C_VEL
LIN {X 0,Y 523.88,Z 1001.151,A -85,B 0,C 180,E1 16251.522,E2 16251.522} C_VEL
LIN {X 0,Y 528.268,Z 982.655,A -85,B 0,C 180,E1 16250.18,E2 16250.18} C_VEL
LIN {X 0,Y 533.632,Z 958.68,A -85,B 0,C 180,E1 16248.663,E2 16248.663} C_VEL
LIN {X 0,Y 538.357,Z 934.714,A -85,B 0,C 180,E1 16247.392,E2 16247.392} C_VEL
LIN {X 0,Y 542.062,Z 914.038,A -85,B 0,C 180,E1 16246.453,E2 16246.453} C_VEL
LIN {X 0,Y 545.395,Z 893.142,A -85,B 0,C 180,E1 16245.643,E2 16245.643} C_VEL
LIN {X 0,Y 548.427,Z 871.19,A -85,B 0,C 180,E1 16244.93,E2 16244.93} C_VEL
LIN {X 0,Y 551.595,Z 843.018,A -85,B 0,C 180,E1 16244.208,E2 16244.208} C_VEL
LIN {X 0,Y 553.601,Z 818.068,A -85,B 0,C 180,E1 16243.74,E2 16243.74} C_VEL
LIN {X 0,Y 561.044,Z 647.729,A -85,B 0,C 180,E1 16241.19,E2 16241.19} C_VEL
LIN {X 0,Y 569.229,Z 463.065,A -85,B 0,C 180,E1 16238.403,E2 16238.403} C_VEL
LIN {X 0,Y 555.964,Z 443.377,A -85,B 0,C 180,E1 16235.895,E2 16235.895} C_VEL
LIN {X 0,Y 545.718,Z 429.564,A -85,B 0,C 180,E1 16233.786,E2 16233.786} C_VEL
LIN {X 0,Y 534.941,Z 415.546,A -85,B 0,C 180,E1 16231.339,E2 16231.339} C_VEL
LIN {X 0,Y 529.182,Z 408.641,A -85,B 0,C 180,E1 16229.923,E2 16229.923} C_VEL
LIN {X 0,Y 525.328,Z 403.822,A -85,B 0,C 180,E1 16228.911,E2 16228.911} C_VEL
LIN {X 0,Y 520.691,Z 398.233,A -85,B 0,C 180,E1 16227.63,E2 16227.63} C_VEL
LIN {X 0,Y 516.898,Z 393.509,A -85,B 0,C 180,E1 16226.511,E2 16226.511} C_VEL
LIN {X 0,Y 512.447,Z 388.571,A -85,B 0,C 180,E1 16225.129,E2 16225.129} C_VEL
LIN {X 0,Y 511.127,Z 386.796,A -85,B 0,C 180,E1 16224.687,E2 16224.687} C_VEL
LIN {X 0,Y 507.55,Z 383.219,A -85,B 0,C 180,E1 16223.481,E2 16223.481} C_VEL
LIN {X 0,Y 506.042,Z 380.81,A -85,B 0,C 180,E1 16222.908,E2 16222.908} C_VEL
LIN {X 0,Y 502.491,Z 377.809,A -85,B 0,C 180,E1 16221.6,E2 16221.6} C_VEL
LIN {X 0,Y 500.44,Z 374.32,A -85,B 0,C 180,E1 16220.711,E2 16220.711} C_VEL
LIN {X 0,Y 496.986,Z 371.924,A -85,B 0,C 180,E1 16219.266,E2 16219.266} C_VEL
LIN {X 0,Y 494.919,Z 368.482,A -85,B 0,C 180,E1 16218.219,E2 16218.219} C_VEL
LIN {X 0,Y 494.553,Z 367.773,A -85,B 0,C 180,E1 16218.019,E2 16218.019} C_VEL
LIN {X 0,Y 491.173,Z 365.826,A -85,B 0,C 180,E1 16216.316,E2 16216.316} C_VEL
LIN {X 0,Y 489.146,Z 362.943,A -85,B 0,C 180,E1 16215.047,E2 16215.047} C_VEL
LIN {X 0,Y 488.381,Z 360.95,A -85,B 0,C 180,E1 16214.464,E2 16214.464} C_VEL
LIN {X 0,Y 484.495,Z 359.02,A -85,B 0,C 180,E1 16211.669,E2 16211.669} C_VEL
LIN {X 0,Y 482.335,Z 355.681,A -85,B 0,C 180,E1 16209.305,E2 16209.305} C_VEL
LIN {X 0,Y 482.042,Z 354.164,A -85,B 0,C 180,E1 16208.709,E2 16208.709} C_VEL
LIN {X 0,Y 481.989,Z 354.17,A -85,B 0,C 180,E1 16205.282,E2 16205.282} C_VEL
LIN {X 0,Y 481.988,Z 354.17,A -85,B 0,C 180,E1 16201.664,E2 16201.664} C_VEL
LIN {X 0,Y 482.038,Z 354.165,A -85,B 0,C 180,E1 16198.336,E2 16198.336} C_VEL
LIN {X 0,Y 481.995,Z 354.305,A -85,B 0,C 180,E1 16197.384,E2 16197.384} C_VEL
LIN {X 0,Y 483.073,Z 357.299,A -85,B 0,C 180,E1 16195.846,E2 16195.846} C_VEL
LIN {X 0,Y 486.252,Z 360.318,A -85,B 0,C 180,E1 16193.032,E2 16193.032} C_VEL
LIN {X 0,Y 488.529,Z 361.309,A -85,B 0,C 180,E1 16191.526,E2 16191.526} C_VEL
LIN {X 0,Y 489.815,Z 364.222,A -85,B 0,C 180,E1 16190.601,E2 16190.601} C_VEL
LIN {X 0,Y 492.418,Z 366.857,A -85,B 0,C 180,E1 16189.115,E2 16189.115} C_VEL
LIN {X 0,Y 494.679,Z 368.057,A -85,B 0,C 180,E1 16188.013,E2 16188.013} C_VEL
LIN {X 0,Y 496.581,Z 371.475,A -85,B 0,C 180,E1 16187.026,E2 16187.026} C_VEL
LIN {X 0,Y 500.088,Z 374.224,A -85,B 0,C 180,E1 16185.527,E2 16185.527} C_VEL
LIN {X 0,Y 500.746,Z 374.98,A -85,B 0,C 180,E1 16185.25,E2 16185.25} C_VEL
LIN {X 0,Y 503.385,Z 378.896,A -85,B 0,C 180,E1 16184.15,E2 16184.15} C_VEL
LIN {X 0,Y 506.374,Z 381.368,A -85,B 0,C 180,E1 16183.067,E2 16183.067} C_VEL
LIN {X 0,Y 509.193,Z 385.263,A -85,B 0,C 180,E1 16182.043,E2 16182.043} C_VEL
LIN {X 0,Y 511.794,Z 387.639,A -85,B 0,C 180,E1 16181.194,E2 16181.194} C_VEL
LIN {X 0,Y 515.228,Z 392.011,A -85,B 0,C 180,E1 16180.087,E2 16180.087} C_VEL
LIN {X 0,Y 517.052,Z 393.868,A -85,B 0,C 180,E1 16179.541,E2 16179.541} C_VEL
LIN {X 0,Y 520.838,Z 398.47,A -85,B 0,C 180,E1 16178.43,E2 16178.43} C_VEL
LIN {X 0,Y 522.75,Z 400.76,A -85,B 0,C 180,E1 16177.893,E2 16177.893} C_VEL
LIN {X 0,Y 527.359,Z 406.33,A -85,B 0,C 180,E1 16176.655,E2 16176.655} C_VEL
LIN {X 0,Y 534.154,Z 414.98,A -85,B 0,C 180,E1 16174.943,E2 16174.943} C_VEL
LIN {X 0,Y 545.237,Z 430.329,A -85,B 0,C 180,E1 16172.386,E2 16172.386} C_VEL
LIN {X 0,Y 556.42,Z 446.584,A -85,B 0,C 180,E1 16170.058,E2 16170.058} C_VEL
LIN {X 0,Y 569.31,Z 466.202,A -85,B 0,C 180,E1 16167.621,E2 16167.621} C_VEL
LIN {X 0,Y 559.788,Z 680.502,A -85,B 0,C 180,E1 16164.404,E2 16164.404} C_VEL
LIN {X 0,Y 553.465,Z 825.745,A -85,B 0,C 180,E1 16162.23,E2 16162.23} C_VEL
LIN {X 0,Y 551.371,Z 851.546,A -85,B 0,C 180,E1 16161.747,E2 16161.747} C_VEL
LIN {X 0,Y 548.197,Z 879.176,A -85,B 0,C 180,E1 16161.039,E2 16161.039} C_VEL
LIN {X 0,Y 545.176,Z 900.893,A -85,B 0,C 180,E1 16160.338,E2 16160.338} C_VEL
LIN {X 0,Y 541.936,Z 921.187,A -85,B 0,C 180,E1 16159.559,E2 16159.559} C_VEL
LIN {X 0,Y 538.263,Z 941.796,A -85,B 0,C 180,E1 16158.631,E2 16158.631} C_VEL
LIN {X 0,Y 533.503,Z 966.035,A -85,B 0,C 180,E1 16157.359,E2 16157.359} C_VEL
LIN {X 0,Y 528.096,Z 990.405,A -85,B 0,C 180,E1 16155.832,E2 16155.832} C_VEL
LIN {X 0,Y 523.69,Z 1009.114,A -85,B 0,C 180,E1 16154.484,E2 16154.484} C_VEL
LIN {X 0,Y 519.299,Z 1026.861,A -85,B 0,C 180,E1 16153.045,E2 16153.045} C_VEL
LIN {X 0,Y 514.86,Z 1044.156,A -85,B 0,C 180,E1 16151.471,E2 16151.471} C_VEL
LIN {X 0,Y 509.622,Z 1064.029,A -85,B 0,C 180,E1 16149.433,E2 16149.433} C_VEL
LIN {X 0,Y 504.215,Z 1083.85,A -85,B 0,C 180,E1 16147.074,E2 16147.074} C_VEL
LIN {X 0,Y 500.084,Z 1099.103,A -85,B 0,C 180,E1 16145.018,E2 16145.018} C_VEL
LIN {X 0,Y 496.434,Z 1112.894,A -85,B 0,C 180,E1 16142.944,E2 16142.944} C_VEL
LIN {X 0,Y 492.896,Z 1126.786,A -85,B 0,C 180,E1 16140.609,E2 16140.609} C_VEL
LIN {X 0,Y 488.868,Z 1143.424,A -85,B 0,C 180,E1 16137.4,E2 16137.4} C_VEL
LIN {X 0,Y 486.295,Z 1155.072,A -85,B 0,C 180,E1 16134.8,E2 16134.8} C_VEL
LIN {X 0,Y 484.364,Z 1164.87,A -85,B 0,C 180,E1 16132.324,E2 16132.324} C_VEL
LIN {X 0,Y 482.806,Z 1173.88,A -85,B 0,C 180,E1 16129.729,E2 16129.729} C_VEL
LIN {X 0,Y 481.434,Z 1183.316,A -85,B 0,C 180,E1 16126.531,E2 16126.531} C_VEL
LIN {X 0,Y 480.634,Z 1190.545,A -85,B 0,C 180,E1 16123.474,E2 16123.474} C_VEL
LIN {X 0,Y 480.227,Z 1195.473,A -85,B 0,C 180,E1 16120.922,E2 16120.922} C_VEL
LIN {X 0,Y 480.03,Z 1199.345,A -85,B 0,C 180,E1 16118.384,E2 16118.384} C_VEL
LIN {X 0,Y 479.94,Z 1202.188,A -85,B 0,C 180,E1 16115.86,E2 16115.86} C_VEL
LIN {X 0,Y 479.916,Z 1204.021,A -85,B 0,C 180,E1 16113.345,E2 16113.345} C_VEL
LIN {X 0,Y 479.898,Z 1204.871,A -85,B 0,C 180,E1 16110.717,E2 16110.717} C_VEL
LIN {X 0,Y 479.909,Z 1204.548,A -85,B 0,C 180,E1 16107.612,E2 16107.612} C_VEL
LIN {X 0,Y 479.936,Z 1202.529,A -85,B 0,C 180,E1 16104.501,E2 16104.501} C_VEL
LIN {X 0,Y 480.019,Z 1199.665,A -85,B 0,C 180,E1 16101.858,E2 16101.858} C_VEL
LIN {X 0,Y 480.205,Z 1195.888,A -85,B 0,C 180,E1 16099.321,E2 16099.321} C_VEL
LIN {X 0,Y 480.581,Z 1191.056,A -85,B 0,C 180,E1 16096.77,E2 16096.77} C_VEL
LIN {X 0,Y 481.215,Z 1185.033,A -85,B 0,C 180,E1 16094.164,E2 16094.164} C_VEL
LIN {X 0,Y 482.446,Z 1176.311,A -85,B 0,C 180,E1 16091.012,E2 16091.012} C_VEL
LIN {X 0,Y 484.188,Z 1165.796,A -85,B 0,C 180,E1 16087.924,E2 16087.924} C_VEL
LIN {X 0,Y 486.133,Z 1155.84,A -85,B 0,C 180,E1 16085.384,E2 16085.384} C_VEL
LIN {X 0,Y 488.472,Z 1145.15,A -85,B 0,C 180,E1 16082.973,E2 16082.973} C_VEL
LIN {X 0,Y 491.524,Z 1132.18,A -85,B 0,C 180,E1 16080.376,E2 16080.376} C_VEL
LIN {X 0,Y 495.85,Z 1115.187,A -85,B 0,C 180,E1 16077.426,E2 16077.426} C_VEL
LIN {X 0,Y 499.628,Z 1100.76,A -85,B 0,C 180,E1 16075.226,E2 16075.226} C_VEL
LIN {X 0,Y 503.704,Z 1085.69,A -85,B 0,C 180,E1 16073.168,E2 16073.168} C_VEL
LIN {X 0,Y 508.333,Z 1068.781,A -85,B 0,C 180,E1 16071.098,E2 16071.098} C_VEL
LIN {X 0,Y 514.614,Z 1045.863,A -85,B 0,C 180,E1 16068.655,E2 16068.655} C_VEL
LIN {X 0,Y 519.388,Z 1027.905,A -85,B 0,C 180,E1 16066.985,E2 16066.985} C_VEL
LIN {X 0,Y 524.075,Z 1009.74,A -85,B 0,C 180,E1 16065.482,E2 16065.482} C_VEL
LIN {X 0,Y 528.832,Z 990.507,A -85,B 0,C 180,E1 16064.072,E2 16064.072} C_VEL
LIN {X 0,Y 534.523,Z 966.205,A -85,B 0,C 180,E1 16062.523,E2 16062.523} C_VEL
LIN {X 0,Y 539.625,Z 941.595,A -85,B 0,C 180,E1 16061.213,E2 16061.213} C_VEL
LIN {X 0,Y 543.409,Z 921.593,A -85,B 0,C 180,E1 16060.3,E2 16060.3} C_VEL
LIN {X 0,Y 546.873,Z 901.256,A -85,B 0,C 180,E1 16059.506,E2 16059.506} C_VEL
LIN {X 0,Y 550.044,Z 879.921,A -85,B 0,C 180,E1 16058.806,E2 16058.806} C_VEL
LIN {X 0,Y 553.398,Z 853.164,A -85,B 0,C 180,E1 16058.103,E2 16058.103} C_VEL
LIN {X 0,Y 555.769,Z 826.08,A -85,B 0,C 180,E1 16057.585,E2 16057.585} C_VEL
LIN {X 0,Y 562.229,Z 694.462,A -85,B 0,C 180,E1 16055.577,E2 16055.577} C_VEL
LIN {X 0,Y 572.994,Z 481.454,A -85,B 0,C 180,E1 16052.321,E2 16052.321} C_VEL
LIN {X 0,Y 573.693,Z 466.848,A -85,B 0,C 180,E1 16052.083,E2 16052.083} C_VEL
LIN {X 0,Y 565.964,Z 454.765,A -85,B 0,C 180,E1 16050.379,E2 16050.379} C_VEL
LIN {X 0,Y 556.641,Z 440.864,A -85,B 0,C 180,E1 16048.128,E2 16048.128} C_VEL
LIN {X 0,Y 549.526,Z 431.148,A -85,B 0,C 180,E1 16046.241,E2 16046.241} C_VEL
LIN {X 0,Y 542.793,Z 421.834,A -85,B 0,C 180,E1 16044.255,E2 16044.255} C_VEL
LIN {X 0,Y 535.849,Z 413.063,A -85,B 0,C 180,E1 16041.971,E2 16041.971} C_VEL
LIN {X 0,Y 532.089,Z 408.671,A -85,B 0,C 180,E1 16040.602,E2 16040.602} C_VEL
LIN {X 0,Y 530.956,Z 407.192,A -85,B 0,C 180,E1 16040.159,E2 16040.159} C_VEL
LIN {X 0,Y 527.468,Z 403.452,A -85,B 0,C 180,E1 16038.742,E2 16038.742} C_VEL
LIN {X 0,Y 526.204,Z 401.406,A -85,B 0,C 180,E1 16038.158,E2 16038.158} C_VEL
LIN {X 0,Y 522.646,Z 398.136,A -85,B 0,C 180,E1 16036.505,E2 16036.505} C_VEL
LIN {X 0,Y 520.82,Z 395.047,A -85,B 0,C 180,E1 16035.477,E2 16035.477} C_VEL
LIN {X 0,Y 517.596,Z 392.712,A -85,B 0,C 180,E1 16033.632,E2 16033.632} C_VEL
LIN {X 0,Y 515.429,Z 388.866,A -85,B 0,C 180,E1 16031.98,E2 16031.98} C_VEL
LIN {X 0,Y 510.989,Z 385.393,A -85,B 0,C 180,E1 16027.533,E2 16027.533} C_VEL
LIN {X 0,Y 509.771,Z 381.957,A -85,B 0,C 180,E1 16023.824,E2 16023.824} C_VEL
LIN {X 0,Y 509.821,Z 382.15,A -85,B 0,C 180,E1 16021.573,E2 16021.573} C_VEL
LIN {X 0,Y 513.073,Z 387.493,A -85,B 0,C 180,E1 16015.753,E2 16015.753} C_VEL
LIN {X 0,Y 515.425,Z 388.846,A -85,B 0,C 180,E1 16013.819,E2 16013.819} C_VEL
LIN {X 0,Y 517.179,Z 392.154,A -85,B 0,C 180,E1 16012.446,E2 16012.446} C_VEL
LIN {X 0,Y 520.484,Z 394.901,A -85,B 0,C 180,E1 16010.49,E2 16010.49} C_VEL
LIN {X 0,Y 521.167,Z 395.678,A -85,B 0,C 180,E1 16010.113,E2 16010.113} C_VEL
LIN {X 0,Y 523.796,Z 399.496,A -85,B 0,C 180,E1 16008.716,E2 16008.716} C_VEL
LIN {X 0,Y 526.514,Z 401.802,A -85,B 0,C 180,E1 16007.497,E2 16007.497} C_VEL
LIN {X 0,Y 529.943,Z 406.301,A -85,B 0,C 180,E1 16006.024,E2 16006.024} C_VEL
LIN {X 0,Y 531.841,Z 408.156,A -85,B 0,C 180,E1 16005.297,E2 16005.297} C_VEL
LIN {X 0,Y 535.462,Z 412.693,A -85,B 0,C 180,E1 16003.956,E2 16003.956} C_VEL
LIN {X 0,Y 537.161,Z 414.672,A -85,B 0,C 180,E1 16003.37,E2 16003.37} C_VEL
LIN {X 0,Y 541.973,Z 420.503,A -85,B 0,C 180,E1 16001.805,E2 16001.805} C_VEL
LIN {X 0,Y 546.69,Z 426.453,A -85,B 0,C 180,E1 16000.39,E2 16000.39} C_VEL
LIN {X 0,Y 551.335,Z 432.38,A -85,B 0,C 180,E1 15999.095,E2 15999.095} C_VEL
LIN {X 0,Y 558.328,Z 441.37,A -85,B 0,C 180,E1 15997.298,E2 15997.298} C_VEL
LIN {X 0,Y 566.233,Z 452.473,A -85,B 0,C 180,E1 15995.426,E2 15995.426} C_VEL
LIN {X 0,Y 573.756,Z 464.127,A -85,B 0,C 180,E1 15993.769,E2 15993.769} C_VEL
LIN {X 0,Y 562.826,Z 678.4,A -85,B 0,C 180,E1 15990.493,E2 15990.493} C_VEL
LIN {X 0,Y 555.923,Z 818.672,A -85,B 0,C 180,E1 15988.352,E2 15988.352} C_VEL
LIN {X 0,Y 553.655,Z 844.902,A -85,B 0,C 180,E1 15987.849,E2 15987.849} C_VEL
LIN {X 0,Y 550.322,Z 872.017,A -85,B 0,C 180,E1 15987.136,E2 15987.136} C_VEL
LIN {X 0,Y 547.18,Z 893.328,A -85,B 0,C 180,E1 15986.434,E2 15986.434} C_VEL
LIN {X 0,Y 543.702,Z 913.902,A -85,B 0,C 180,E1 15985.626,E2 15985.626} C_VEL
LIN {X 0,Y 539.717,Z 934.887,A -85,B 0,C 180,E1 15984.662,E2 15984.662} C_VEL
LIN {X 0,Y 534.408,Z 960.14,A -85,B 0,C 180,E1 15983.294,E2 15983.294} C_VEL
LIN {X 0,Y 529.066,Z 982.837,A -85,B 0,C 180,E1 15981.829,E2 15981.829} C_VEL
LIN {X 0,Y 524.246,Z 1002.164,A -85,B 0,C 180,E1 15980.401,E2 15980.401} C_VEL
LIN {X 0,Y 519.291,Z 1021.144,A -85,B 0,C 180,E1 15978.813,E2 15978.813} C_VEL
LIN {X 0,Y 513.116,Z 1043.944,A -85,B 0,C 180,E1 15976.621,E2 15976.621} C_VEL
LIN {X 0,Y 508.102,Z 1061.914,A -85,B 0,C 180,E1 15974.629,E2 15974.629} C_VEL
LIN {X 0,Y 503.728,Z 1077.629,A -85,B 0,C 180,E1 15972.676,E2 15972.676} C_VEL
LIN {X 0,Y 500.026,Z 1091.07,A -85,B 0,C 180,E1 15970.823,E2 15970.823} C_VEL
LIN {X 0,Y 497.867,Z 1096.042,A -85,B 0,C 180,E1 15970.174,E2 15970.174} C_VEL
LIN {X 0,Y 488.835,Z 1109.04,A -85,B 0,C 180,E1 15968.531,E2 15968.531} C_VEL
LIN {X 0,Y 487.097,Z 1112.775,A -85,B 0,C 180,E1 15967.922,E2 15967.922} C_VEL
LIN {X 0,Y 483.635,Z 1125.697,A -85,B 0,C 180,E1 15965.516,E2 15965.516} C_VEL
LIN {X 0,Y 480.794,Z 1136.981,A -85,B 0,C 180,E1 15963.157,E2 15963.157} C_VEL
LIN {X 0,Y 478.204,Z 1148.16,A -85,B 0,C 180,E1 15960.518,E2 15960.518} C_VEL
LIN {X 0,Y 475.681,Z 1160.457,A -85,B 0,C 180,E1 15957.137,E2 15957.137} C_VEL
LIN {X 0,Y 474.149,Z 1169.189,A -85,B 0,C 180,E1 15954.28,E2 15954.28} C_VEL
LIN {X 0,Y 473.216,Z 1175.929,A -85,B 0,C 180,E1 15951.701,E2 15951.701} C_VEL
LIN {X 0,Y 472.548,Z 1181.862,A -85,B 0,C 180,E1 15949.017,E2 15949.017} C_VEL
LIN {X 0,Y 472.177,Z 1186.864,A -85,B 0,C 180,E1 15946.231,E2 15946.231} C_VEL
LIN {X 0,Y 471.971,Z 1191.215,A -85,B 0,C 180,E1 15942.958,E2 15942.958} C_VEL
LIN {X 0,Y 471.915,Z 1193.655,A -85,B 0,C 180,E1 15940.005,E2 15940.005} C_VEL
LIN {X 0,Y 471.915,Z 1194.732,A -85,B 0,C 180,E1 15937.425,E2 15937.425} C_VEL
LIN {X 0,Y 471.903,Z 1194.826,A -85,B 0,C 180,E1 15934.983,E2 15934.983} C_VEL
LIN {X 0,Y 471.914,Z 1194.016,A -85,B 0,C 180,E1 15932.55,E2 15932.55} C_VEL
LIN {X 0,Y 471.954,Z 1192.188,A -85,B 0,C 180,E1 15930,E2 15930} C_VEL
LIN {X 0,Y 472.039,Z 1189.372,A -85,B 0,C 180,E1 15927.45,E2 15927.45} C_VEL
LIN {X 0,Y 472.242,Z 1185.558,A -85,B 0,C 180,E1 15924.898,E2 15924.898} C_VEL
LIN {X 0,Y 472.671,Z 1180.73,A -85,B 0,C 180,E1 15922.341,E2 15922.341} C_VEL
LIN {X 0,Y 473.608,Z 1173.131,A -85,B 0,C 180,E1 15919.046,E2 15919.046} C_VEL
LIN {X 0,Y 475.016,Z 1163.95,A -85,B 0,C 180,E1 15915.867,E2 15915.867} C_VEL
LIN {X 0,Y 476.662,Z 1155.313,A -85,B 0,C 180,E1 15913.298,E2 15913.298} C_VEL
LIN {X 0,Y 478.787,Z 1145.443,A -85,B 0,C 180,E1 15910.727,E2 15910.727} C_VEL
LIN {X 0,Y 481.702,Z 1133.23,A -85,B 0,C 180,E1 15907.932,E2 15907.932} C_VEL
LIN {X 0,Y 485.71,Z 1117.886,A -85,B 0,C 180,E1 15904.908,E2 15904.908} C_VEL
LIN {X 0,Y 489.505,Z 1103.946,A -85,B 0,C 180,E1 15902.507,E2 15902.507} C_VEL
LIN {X 0,Y 493.456,Z 1090.005,A -85,B 0,C 180,E1 15900.369,E2 15900.369} C_VEL
LIN {X 0,Y 497.896,Z 1074.53,A -85,B 0,C 180,E1 15898.254,E2 15898.254} C_VEL
LIN {X 0,Y 503.815,Z 1053.836,A -85,B 0,C 180,E1 15895.782,E2 15895.782} C_VEL
LIN {X 0,Y 508.895,Z 1035.481,A -85,B 0,C 180,E1 15893.882,E2 15893.882} C_VEL
LIN {X 0,Y 513.49,Z 1018.358,A -85,B 0,C 180,E1 15892.307,E2 15892.307} C_VEL
LIN {X 0,Y 518.034,Z 1000.745,A -85,B 0,C 180,E1 15890.864,E2 15890.864} C_VEL
LIN {X 0,Y 522.837,Z 981.115,A -85,B 0,C 180,E1 15889.442,E2 15889.442} C_VEL
LIN {X 0,Y 528.72,Z 955.125,A -85,B 0,C 180,E1 15887.828,E2 15887.828} C_VEL
LIN {X 0,Y 533.03,Z 933.793,A -85,B 0,C 180,E1 15886.705,E2 15886.705} C_VEL
LIN {X 0,Y 536.826,Z 913.121,A -85,B 0,C 180,E1 15885.77,E2 15885.77} C_VEL
LIN {X 0,Y 540.228,Z 892.319,A -85,B 0,C 180,E1 15884.969,E2 15884.969} C_VEL
LIN {X 0,Y 543.546,Z 868.807,A -85,B 0,C 180,E1 15884.214,E2 15884.214} C_VEL
LIN {X 0,Y 546.704,Z 840.345,A -85,B 0,C 180,E1 15883.507,E2 15883.507} C_VEL
LIN {X 0,Y 548.578,Z 817.183,A -85,B 0,C 180,E1 15883.079,E2 15883.079} C_VEL
LIN {X 0,Y 557.705,Z 615.307,A -85,B 0,C 180,E1 15880.044,E2 15880.044} C_VEL
LIN {X 0,Y 564.512,Z 467.362,A -85,B 0,C 180,E1 15877.796,E2 15877.796} C_VEL
LIN {X 0,Y 552.585,Z 449.5,A -85,B 0,C 180,E1 15875.481,E2 15875.481} C_VEL
LIN {X 0,Y 540.74,Z 433.323,A -85,B 0,C 180,E1 15872.964,E2 15872.964} C_VEL
LIN {X 0,Y 530.924,Z 420.843,A -85,B 0,C 180,E1 15870.658,E2 15870.658} C_VEL
LIN {X 0,Y 526.97,Z 415.925,A -85,B 0,C 180,E1 15869.655,E2 15869.655} C_VEL
LIN {X 0,Y 522.866,Z 410.809,A -85,B 0,C 180,E1 15868.56,E2 15868.56} C_VEL
LIN {X 0,Y 518.477,Z 405.441,A -85,B 0,C 180,E1 15867.322,E2 15867.322} C_VEL
LIN {X 0,Y 513.959,Z 399.934,A -85,B 0,C 180,E1 15865.959,E2 15865.959} C_VEL
LIN {X 0,Y 510.239,Z 395.545,A -85,B 0,C 180,E1 15864.764,E2 15864.764} C_VEL
LIN {X 0,Y 509.043,Z 394.135,A -85,B 0,C 180,E1 15864.362,E2 15864.362} C_VEL
LIN {X 0,Y 505.4,Z 390.177,A -85,B 0,C 180,E1 15863.093,E2 15863.093} C_VEL
LIN {X 0,Y 504.189,Z 388.345,A -85,B 0,C 180,E1 15862.627,E2 15862.627} C_VEL
LIN {X 0,Y 500.576,Z 385.021,A -85,B 0,C 180,E1 15861.257,E2 15861.257} C_VEL
LIN {X 0,Y 498.67,Z 381.951,A -85,B 0,C 180,E1 15860.42,E2 15860.42} C_VEL
LIN {X 0,Y 495.304,Z 379.349,A -85,B 0,C 180,E1 15858.967,E2 15858.967} C_VEL
LIN {X 0,Y 493.13,Z 375.594,A -85,B 0,C 180,E1 15857.829,E2 15857.829} C_VEL
LIN {X 0,Y 489.813,Z 373.539,A -85,B 0,C 180,E1 15856.119,E2 15856.119} C_VEL
LIN {X 0,Y 487.738,Z 370.508,A -85,B 0,C 180,E1 15854.787,E2 15854.787} C_VEL
LIN {X 0,Y 487.055,Z 368.819,A -85,B 0,C 180,E1 15854.262,E2 15854.262} C_VEL
LIN {X 0,Y 483.139,Z 366.657,A -85,B 0,C 180,E1 15851.339,E2 15851.339} C_VEL
LIN {X 0,Y 481.188,Z 363.382,A -85,B 0,C 180,E1 15849.087,E2 15849.087} C_VEL
LIN {X 0,Y 480.852,Z 362.073,A -85,B 0,C 180,E1 15848.49,E2 15848.49} C_VEL
LIN {X 0,Y 478.947,Z 361.571,A -85,B 0,C 180,E1 15841.555,E2 15841.555} C_VEL
LIN {X 0,Y 480.911,Z 362.335,A -85,B 0,C 180,E1 15837.498,E2 15837.498} C_VEL
LIN {X 0,Y 482.52,Z 365.998,A -85,B 0,C 180,E1 15835.364,E2 15835.364} C_VEL
LIN {X 0,Y 485.949,Z 368.556,A -85,B 0,C 180,E1 15832.552,E2 15832.552} C_VEL
LIN {X 0,Y 487.184,Z 369.149,A -85,B 0,C 180,E1 15831.74,E2 15831.74} C_VEL
LIN {X 0,Y 488.821,Z 372.407,A -85,B 0,C 180,E1 15830.582,E2 15830.582} C_VEL
LIN {X 0,Y 491.451,Z 374.856,A -85,B 0,C 180,E1 15829.093,E2 15829.093} C_VEL
LIN {X 0,Y 493.174,Z 375.806,A -85,B 0,C 180,E1 15828.243,E2 15828.243} C_VEL
LIN {X 0,Y 495.355,Z 379.429,A -85,B 0,C 180,E1 15827.112,E2 15827.112} C_VEL
LIN {X 0,Y 499.032,Z 382.467,A -85,B 0,C 180,E1 15825.525,E2 15825.525} C_VEL
LIN {X 0,Y 501.839,Z 386.574,A -85,B 0,C 180,E1 15824.337,E2 15824.337} C_VEL
LIN {X 0,Y 504.639,Z 388.995,A -85,B 0,C 180,E1 15823.303,E2 15823.303} C_VEL
LIN {X 0,Y 507.747,Z 393.1,A -85,B 0,C 180,E1 15822.168,E2 15822.168} C_VEL
LIN {X 0,Y 509.992,Z 395.272,A -85,B 0,C 180,E1 15821.422,E2 15821.422} C_VEL
LIN {X 0,Y 513.572,Z 399.697,A -85,B 0,C 180,E1 15820.257,E2 15820.257} C_VEL
LIN {X 0,Y 515.193,Z 401.508,A -85,B 0,C 180,E1 15819.76,E2 15819.76} C_VEL
LIN {X 0,Y 519.139,Z 406.163,A -85,B 0,C 180,E1 15818.593,E2 15818.593} C_VEL
LIN {X 0,Y 525.312,Z 413.837,A -85,B 0,C 180,E1 15816.885,E2 15816.885} C_VEL
LIN {X 0,Y 531.843,Z 422.263,A -85,B 0,C 180,E1 15815.213,E2 15815.213} C_VEL
LIN {X 0,Y 542.601,Z 437.349,A -85,B 0,C 180,E1 15812.687,E2 15812.687} C_VEL
LIN {X 0,Y 553.555,Z 453.5,A -85,B 0,C 180,E1 15810.365,E2 15810.365} C_VEL
LIN {X 0,Y 564.585,Z 470.49,A -85,B 0,C 180,E1 15808.228,E2 15808.228} C_VEL
LIN {X 0,Y 554.753,Z 684.325,A -85,B 0,C 180,E1 15805.003,E2 15805.003} C_VEL
LIN {X 0,Y 548.37,Z 825.754,A -85,B 0,C 180,E1 15802.874,E2 15802.874} C_VEL
LIN {X 0,Y 546.171,Z 852.08,A -85,B 0,C 180,E1 15802.379,E2 15802.379} C_VEL
LIN {X 0,Y 542.915,Z 879.441,A -85,B 0,C 180,E1 15801.673,E2 15801.673} C_VEL
LIN {X 0,Y 539.929,Z 900.326,A -85,B 0,C 180,E1 15800.999,E2 15800.999} C_VEL
LIN {X 0,Y 536.516,Z 921.119,A -85,B 0,C 180,E1 15800.201,E2 15800.201} C_VEL
LIN {X 0,Y 532.598,Z 942.429,A -85,B 0,C 180,E1 15799.238,E2 15799.238} C_VEL
LIN {X 0,Y 527.5,Z 967.437,A -85,B 0,C 180,E1 15797.91,E2 15797.91} C_VEL
LIN {X 0,Y 522.261,Z 990.271,A -85,B 0,C 180,E1 15796.465,E2 15796.465} C_VEL
LIN {X 0,Y 517.581,Z 1009.474,A -85,B 0,C 180,E1 15795.074,E2 15795.074} C_VEL
LIN {X 0,Y 513.039,Z 1027.202,A -85,B 0,C 180,E1 15793.624,E2 15793.624} C_VEL
LIN {X 0,Y 508.194,Z 1045.401,A -85,B 0,C 180,E1 15791.95,E2 15791.95} C_VEL
LIN {X 0,Y 502.215,Z 1067.064,A -85,B 0,C 180,E1 15789.671,E2 15789.671} C_VEL
LIN {X 0,Y 497.254,Z 1084.629,A -85,B 0,C 180,E1 15787.537,E2 15787.537} C_VEL
LIN {X 0,Y 493.208,Z 1098.996,A -85,B 0,C 180,E1 15785.58,E2 15785.58} C_VEL
LIN {X 0,Y 489.377,Z 1112.796,A -85,B 0,C 180,E1 15783.481,E2 15783.481} C_VEL
LIN {X 0,Y 485.583,Z 1126.992,A -85,B 0,C 180,E1 15781.062,E2 15781.062} C_VEL
LIN {X 0,Y 481.413,Z 1143.329,A -85,B 0,C 180,E1 15777.861,E2 15777.861} C_VEL
LIN {X 0,Y 478.708,Z 1154.979,A -85,B 0,C 180,E1 15775.22,E2 15775.22} C_VEL
LIN {X 0,Y 476.665,Z 1164.777,A -85,B 0,C 180,E1 15772.704,E2 15772.704} C_VEL
LIN {X 0,Y 474.934,Z 1174.197,A -85,B 0,C 180,E1 15769.942,E2 15769.942} C_VEL
LIN {X 0,Y 473.412,Z 1184.193,A -85,B 0,C 180,E1 15766.441,E2 15766.441} C_VEL
LIN {X 0,Y 472.691,Z 1190.542,A -85,B 0,C 180,E1 15763.705,E2 15763.705} C_VEL
LIN {X 0,Y 472.249,Z 1195.47,A -85,B 0,C 180,E1 15761.109,E2 15761.109} C_VEL
LIN {X 0,Y 472.048,Z 1199.183,A -85,B 0,C 180,E1 15758.65,E2 15758.65} C_VEL
LIN {X 0,Y 471.95,Z 1201.958,A -85,B 0,C 180,E1 15756.203,E2 15756.203} C_VEL
LIN {X 0,Y 471.915,Z 1203.872,A -85,B 0,C 180,E1 15753.663,E2 15753.663} C_VEL
LIN {X 0,Y 471.913,Z 1204.78,A -85,B 0,C 180,E1 15751.215,E2 15751.215} C_VEL
LIN {X 0,Y 471.913,Z 1204.78,A -85,B 0,C 180,E1 15748.786,E2 15748.786} C_VEL
LIN {X 0,Y 471.914,Z 1203.871,A -85,B 0,C 180,E1 15746.338,E2 15746.338} C_VEL
LIN {X 0,Y 471.949,Z 1201.957,A -85,B 0,C 180,E1 15743.798,E2 15743.798} C_VEL
LIN {X 0,Y 472.056,Z 1199.023,A -85,B 0,C 180,E1 15741.228,E2 15741.228} C_VEL
LIN {X 0,Y 472.296,Z 1194.852,A -85,B 0,C 180,E1 15738.522,E2 15738.522} C_VEL
LIN {X 0,Y 472.951,Z 1188.164,A -85,B 0,C 180,E1 15735.179,E2 15735.179} C_VEL
LIN {X 0,Y 473.92,Z 1180.493,A -85,B 0,C 180,E1 15732.187,E2 15732.187} C_VEL
LIN {X 0,Y 475.206,Z 1172.559,A -85,B 0,C 180,E1 15729.557,E2 15729.557} C_VEL
LIN {X 0,Y 476.885,Z 1163.659,A -85,B 0,C 180,E1 15726.994,E2 15726.994} C_VEL
LIN {X 0,Y 479.307,Z 1152.378,A -85,B 0,C 180,E1 15724.152,E2 15724.152} C_VEL
LIN {X 0,Y 482.786,Z 1137.835,A -85,B 0,C 180,E1 15721.013,E2 15721.013} C_VEL
LIN {X 0,Y 486.177,Z 1124.541,A -85,B 0,C 180,E1 15718.509,E2 15718.509} C_VEL
LIN {X 0,Y 489.793,Z 1111.203,A -85,B 0,C 180,E1 15716.272,E2 15716.272} C_VEL
LIN {X 0,Y 494.532,Z 1094.531,A -85,B 0,C 180,E1 15713.779,E2 15713.779} C_VEL
LIN {X 0,Y 500.1,Z 1075.019,A -85,B 0,C 180,E1 15711.239,E2 15711.239} C_VEL
LIN {X 0,Y 505.027,Z 1057.791,A -85,B 0,C 180,E1 15709.265,E2 15709.265} C_VEL
LIN {X 0,Y 509.749,Z 1041.149,A -85,B 0,C 180,E1 15707.565,E2 15707.565} C_VEL
LIN {X 0,Y 514.705,Z 1023.272,A -85,B 0,C 180,E1 15705.937,E2 15705.937} C_VEL
LIN {X 0,Y 520.812,Z 1000.415,A -85,B 0,C 180,E1 15704.11,E2 15704.11} C_VEL
LIN {X 0,Y 526.492,Z 977.265,A -85,B 0,C 180,E1 15702.536,E2 15702.536} C_VEL
LIN {X 0,Y 530.946,Z 958.006,A -85,B 0,C 180,E1 15701.4,E2 15701.4} C_VEL
LIN {X 0,Y 535.023,Z 938.725,A -85,B 0,C 180,E1 15700.399,E2 15700.399} C_VEL
LIN {X 0,Y 538.964,Z 918.362,A -85,B 0,C 180,E1 15699.489,E2 15699.489} C_VEL
LIN {X 0,Y 543.173,Z 893.904,A -85,B 0,C 180,E1 15698.568,E2 15698.568} C_VEL
LIN {X 0,Y 546.988,Z 866.681,A -85,B 0,C 180,E1 15697.76,E2 15697.76} C_VEL
LIN {X 0,Y 549.504,Z 844.569,A -85,B 0,C 180,E1 15697.25,E2 15697.25} C_VEL
LIN {X 0,Y 551.368,Z 822.329,A -85,B 0,C 180,E1 15696.845,E2 15696.845} C_VEL
LIN {X 0,Y 562.332,Z 606.309,A -85,B 0,C 180,E1 15693.541,E2 15693.541} C_VEL
LIN {X 0,Y 569.503,Z 471.399,A -85,B 0,C 180,E1 15691.459,E2 15691.459} C_VEL
LIN {X 0,Y 562.043,Z 459.661,A -85,B 0,C 180,E1 15689.756,E2 15689.756} C_VEL
LIN {X 0,Y 553.16,Z 446.322,A -85,B 0,C 180,E1 15687.535,E2 15687.535} C_VEL
LIN {X 0,Y 544.274,Z 433.973,A -85,B 0,C 180,E1 15685.053,E2 15685.053} C_VEL
LIN {X 0,Y 538.187,Z 425.709,A -85,B 0,C 180,E1 15683.138,E2 15683.138} C_VEL
LIN {X 0,Y 533.858,Z 420.363,A -85,B 0,C 180,E1 15681.652,E2 15681.652} C_VEL
LIN {X 0,Y 530.121,Z 415.734,A -85,B 0,C 180,E1 15680.25,E2 15680.25} C_VEL
LIN {X 0,Y 525.665,Z 410.65,A -85,B 0,C 180,E1 15678.407,E2 15678.407} C_VEL
LIN {X 0,Y 524.52,Z 408.981,A -85,B 0,C 180,E1 15677.873,E2 15677.873} C_VEL
LIN {X 0,Y 520.958,Z 405.416,A -85,B 0,C 180,E1 15676.159,E2 15676.159} C_VEL
LIN {X 0,Y 519.249,Z 402.746,A -85,B 0,C 180,E1 15675.182,E2 15675.182} C_VEL
LIN {X 0,Y 516.056,Z 400.115,A -85,B 0,C 180,E1 15673.274,E2 15673.274} C_VEL
LIN {X 0,Y 514.044,Z 396.426,A -85,B 0,C 180,E1 15671.671,E2 15671.671} C_VEL
LIN {X 0,Y 510.079,Z 393.525,A -85,B 0,C 180,E1 15667.66,E2 15667.66} C_VEL
LIN {X 0,Y 508.795,Z 389.898,A -85,B 0,C 180,E1 15663.831,E2 15663.831} C_VEL
LIN {X 0,Y 508.836,Z 390.15,A -85,B 0,C 180,E1 15661.576,E2 15661.576} C_VEL
LIN {X 0,Y 512.096,Z 395.453,A -85,B 0,C 180,E1 15655.745,E2 15655.745} C_VEL
LIN {X 0,Y 514.223,Z 396.71,A -85,B 0,C 180,E1 15653.973,E2 15653.973} C_VEL
LIN {X 0,Y 516.193,Z 400.231,A -85,B 0,C 180,E1 15652.431,E2 15652.431} C_VEL
LIN {X 0,Y 519.695,Z 403.208,A -85,B 0,C 180,E1 15650.364,E2 15650.364} C_VEL
LIN {X 0,Y 522.372,Z 407.175,A -85,B 0,C 180,E1 15648.909,E2 15648.909} C_VEL
LIN {X 0,Y 525.046,Z 409.537,A -85,B 0,C 180,E1 15647.685,E2 15647.685} C_VEL
LIN {X 0,Y 528.569,Z 414.098,A -85,B 0,C 180,E1 15646.155,E2 15646.155} C_VEL
LIN {X 0,Y 530.301,Z 415.92,A -85,B 0,C 180,E1 15645.477,E2 15645.477} C_VEL
LIN {X 0,Y 534.043,Z 420.502,A -85,B 0,C 180,E1 15644.08,E2 15644.08} C_VEL
LIN {X 0,Y 540.173,Z 428.071,A -85,B 0,C 180,E1 15642.021,E2 15642.021} C_VEL
LIN {X 0,Y 544.92,Z 434.142,A -85,B 0,C 180,E1 15640.574,E2 15640.574} C_VEL
LIN {X 0,Y 549.522,Z 440.081,A -85,B 0,C 180,E1 15639.274,E2 15639.274} C_VEL
LIN {X 0,Y 556.543,Z 449.304,A -85,B 0,C 180,E1 15637.444,E2 15637.444} C_VEL
LIN {X 0,Y 563.681,Z 459.486,A -85,B 0,C 180,E1 15635.726,E2 15635.726} C_VEL
LIN {X 0,Y 569.537,Z 468.689,A -85,B 0,C 180,E1 15634.399,E2 15634.399} C_VEL
LIN {X 0,Y 558.154,Z 684.283,A -85,B 0,C 180,E1 15631.092,E2 15631.092} C_VEL
LIN {X 0,Y 551.282,Z 818.822,A -85,B 0,C 180,E1 15629.028,E2 15629.028} C_VEL
LIN {X 0,Y 548.902,Z 845.483,A -85,B 0,C 180,E1 15628.515,E2 15628.515} C_VEL
LIN {X 0,Y 545.468,Z 872.402,A -85,B 0,C 180,E1 15627.804,E2 15627.804} C_VEL
LIN {X 0,Y 542.312,Z 893.178,A -85,B 0,C 180,E1 15627.12,E2 15627.12} C_VEL
LIN {X 0,Y 538.811,Z 913.286,A -85,B 0,C 180,E1 15626.333,E2 15626.333} C_VEL
LIN {X 0,Y 534.924,Z 933.195,A -85,B 0,C 180,E1 15625.423,E2 15625.423} C_VEL
LIN {X 0,Y 530.497,Z 953.895,A -85,B 0,C 180,E1 15624.325,E2 15624.325} C_VEL
LIN {X 0,Y 524.698,Z 978.503,A -85,B 0,C 180,E1 15622.801,E2 15622.801} C_VEL
LIN {X 0,Y 519.198,Z 999.785,A -85,B 0,C 180,E1 15621.252,E2 15621.252} C_VEL
LIN {X 0,Y 514.259,Z 1018.033,A -85,B 0,C 180,E1 15619.741,E2 15619.741} C_VEL
LIN {X 0,Y 509.435,Z 1035.237,A -85,B 0,C 180,E1 15618.138,E2 15618.138} C_VEL
LIN {X 0,Y 504.161,Z 1053.62,A -85,B 0,C 180,E1 15616.211,E2 15616.211} C_VEL
LIN {X 0,Y 498.004,Z 1074.561,A -85,B 0,C 180,E1 15613.683,E2 15613.683} C_VEL
LIN {X 0,Y 493.407,Z 1090.354,A -85,B 0,C 180,E1 15611.502,E2 15611.502} C_VEL
LIN {X 0,Y 489.243,Z 1105.026,A -85,B 0,C 180,E1 15609.233,E2 15609.233} C_VEL
LIN {X 0,Y 487.097,Z 1112.775,A -85,B 0,C 180,E1 15607.922,E2 15607.922} C_VEL
LIN {X 0,Y 485.008,Z 1117.161,A -85,B 0,C 180,E1 15607.205,E2 15607.205} C_VEL
LIN {X 0,Y 476.282,Z 1128.883,A -85,B 0,C 180,E1 15605.368,E2 15605.368} C_VEL
LIN {X 0,Y 474.67,Z 1132.224,A -85,B 0,C 180,E1 15604.701,E2 15604.701} C_VEL
LIN {X 0,Y 471.35,Z 1145.149,A -85,B 0,C 180,E1 15601.717,E2 15601.717} C_VEL
LIN {X 0,Y 469.054,Z 1155.172,A -85,B 0,C 180,E1 15599.072,E2 15599.072} C_VEL
LIN {X 0,Y 467.205,Z 1164.348,A -85,B 0,C 180,E1 15596.295,E2 15596.295} C_VEL
LIN {X 0,Y 465.572,Z 1174.209,A -85,B 0,C 180,E1 15592.741,E2 15592.741} C_VEL
LIN {X 0,Y 464.741,Z 1180.663,A -85,B 0,C 180,E1 15589.872,E2 15589.872} C_VEL
LIN {X 0,Y 464.294,Z 1185.439,A -85,B 0,C 180,E1 15587.288,E2 15587.288} C_VEL
LIN {X 0,Y 464.059,Z 1189.302,A -85,B 0,C 180,E1 15584.659,E2 15584.659} C_VEL
LIN {X 0,Y 463.944,Z 1192.136,A -85,B 0,C 180,E1 15582.066,E2 15582.066} C_VEL
LIN {X 0,Y 463.915,Z 1193.939,A -85,B 0,C 180,E1 15579.552,E2 15579.552} C_VEL
LIN {X 0,Y 463.905,Z 1194.805,A -85,B 0,C 180,E1 15577.056,E2 15577.056} C_VEL
LIN {X 0,Y 463.905,Z 1194.753,A -85,B 0,C 180,E1 15574.574,E2 15574.574} C_VEL
LIN {X 0,Y 463.92,Z 1193.798,A -85,B 0,C 180,E1 15572.099,E2 15572.099} C_VEL
LIN {X 0,Y 463.962,Z 1191.829,A -85,B 0,C 180,E1 15569.506,E2 15569.506} C_VEL
LIN {X 0,Y 464.083,Z 1188.712,A -85,B 0,C 180,E1 15566.788,E2 15566.788} C_VEL
